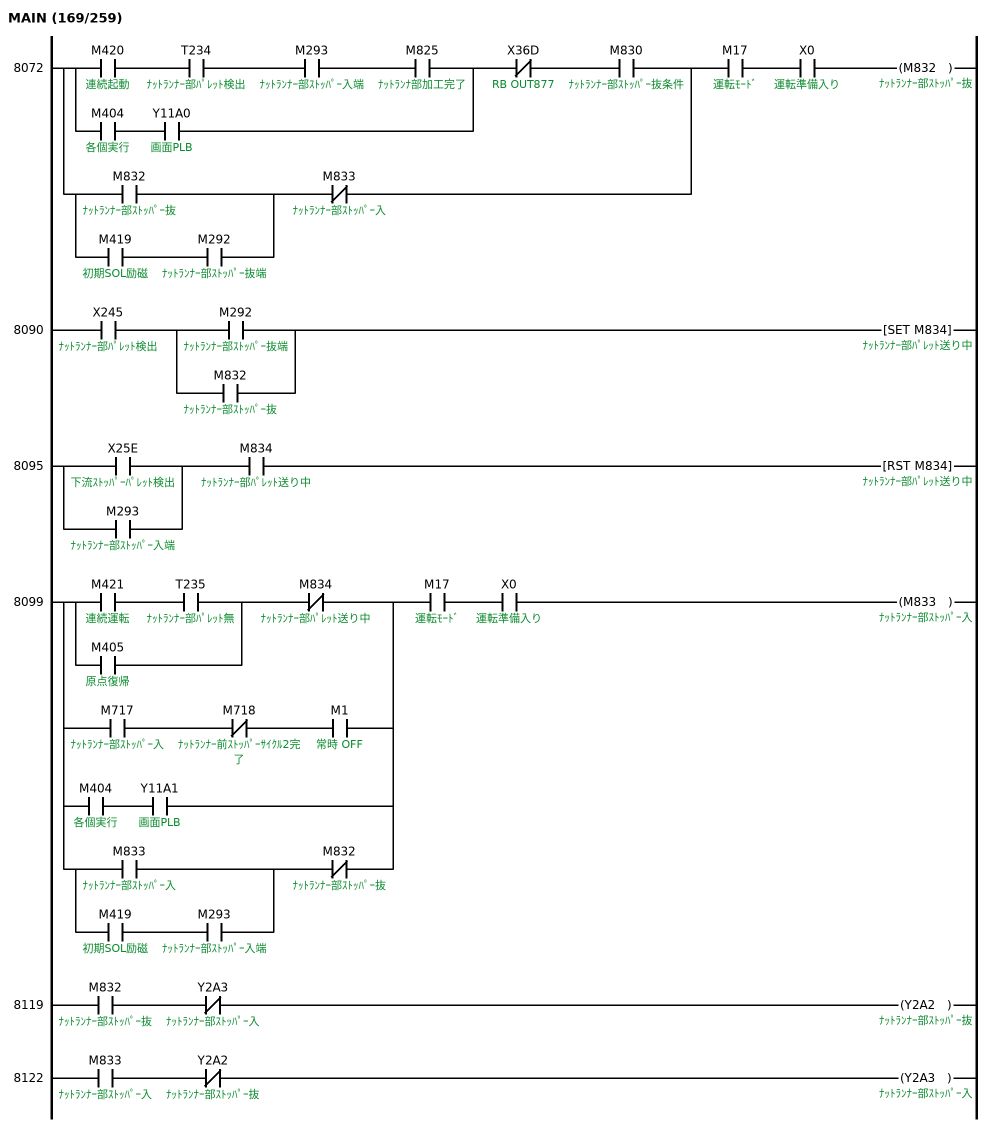
[picture p168: ladder of MAIN, rungs at steps 8072 to 8122]
8072  LD      M420  ; 連続起動
      AND     T234  ; ﾅｯﾄﾗﾝﾅｰ部ﾊﾟﾚｯﾄ検出
      AND     M293  ; ﾅｯﾄﾗﾝﾅｰ部ｽﾄｯﾊﾟｰ入端
      AND     M825  ; ﾅｯﾄﾗﾝﾅ部加工完了
      LD      M404  ; 各個実行
      AND     Y11A0  ; 画面PLB
      ORB
      ANI     X36D  ; RB OUT877
      AND     M830  ; ﾅｯﾄﾗﾝﾅｰ部ｽﾄｯﾊﾟｰ抜条件
      LD      M832  ; ﾅｯﾄﾗﾝﾅｰ部ｽﾄｯﾊﾟｰ抜
      LD      M419  ; 初期SOL励磁
      AND     M292  ; ﾅｯﾄﾗﾝﾅｰ部ｽﾄｯﾊﾟｰ抜端
      ORB
      ANI     M833  ; ﾅｯﾄﾗﾝﾅｰ部ｽﾄｯﾊﾟｰ入
      ORB
      AND     M17  ; 運転ﾓｰﾄﾞ
      AND     X0  ; 運転準備入り
      OUT     M832  ; ﾅｯﾄﾗﾝﾅｰ部ｽﾄｯﾊﾟｰ抜
8090  LD      X245  ; ﾅｯﾄﾗﾝﾅｰ部ﾊﾟﾚｯﾄ検出
      LD      M292  ; ﾅｯﾄﾗﾝﾅｰ部ｽﾄｯﾊﾟｰ抜端
      OR      M832  ; ﾅｯﾄﾗﾝﾅｰ部ｽﾄｯﾊﾟｰ抜
      ANB
      SET     M834  ; ﾅｯﾄﾗﾝﾅｰ部ﾊﾟﾚｯﾄ送り中
8095  LD      X25E  ; 下流ｽﾄｯﾊﾟｰﾊﾟﾚｯﾄ検出
      OR      M293  ; ﾅｯﾄﾗﾝﾅｰ部ｽﾄｯﾊﾟｰ入端
      AND     M834  ; ﾅｯﾄﾗﾝﾅｰ部ﾊﾟﾚｯﾄ送り中
      RST     M834  ; ﾅｯﾄﾗﾝﾅｰ部ﾊﾟﾚｯﾄ送り中
8099  LD      M421  ; 連続運転
      AND     T235  ; ﾅｯﾄﾗﾝﾅｰ部ﾊﾟﾚｯﾄ無
      OR      M405  ; 原点復帰
      ANI     M834  ; ﾅｯﾄﾗﾝﾅｰ部ﾊﾟﾚｯﾄ送り中
      LD      M717  ; ﾅｯﾄﾗﾝﾅｰ部ｽﾄｯﾊﾟｰ入
      ANI     M718  ; ﾅｯﾄﾗﾝﾅｰ前ｽﾄｯﾊﾟｰｻｲｸﾙ2完了
      AND     M1  ; 常時 OFF
      ORB
      LD      M404  ; 各個実行
      AND     Y11A1  ; 画面PLB
      ORB
      LD      M833  ; ﾅｯﾄﾗﾝﾅｰ部ｽﾄｯﾊﾟｰ入
      LD      M419  ; 初期SOL励磁
      AND     M293  ; ﾅｯﾄﾗﾝﾅｰ部ｽﾄｯﾊﾟｰ入端
      ORB
      ANI     M832  ; ﾅｯﾄﾗﾝﾅｰ部ｽﾄｯﾊﾟｰ抜
      ORB
      AND     M17  ; 運転ﾓｰﾄﾞ
      AND     X0  ; 運転準備入り
      OUT     M833  ; ﾅｯﾄﾗﾝﾅｰ部ｽﾄｯﾊﾟｰ入
8119  LD      M832  ; ﾅｯﾄﾗﾝﾅｰ部ｽﾄｯﾊﾟｰ抜
      ANI     Y2A3  ; ﾅｯﾄﾗﾝﾅｰ部ｽﾄｯﾊﾟｰ入
      OUT     Y2A2  ; ﾅｯﾄﾗﾝﾅｰ部ｽﾄｯﾊﾟｰ抜
8122  LD      M833  ; ﾅｯﾄﾗﾝﾅｰ部ｽﾄｯﾊﾟｰ入
      ANI     Y2A2  ; ﾅｯﾄﾗﾝﾅｰ部ｽﾄｯﾊﾟｰ抜
      OUT     Y2A3  ; ﾅｯﾄﾗﾝﾅｰ部ｽﾄｯﾊﾟｰ入
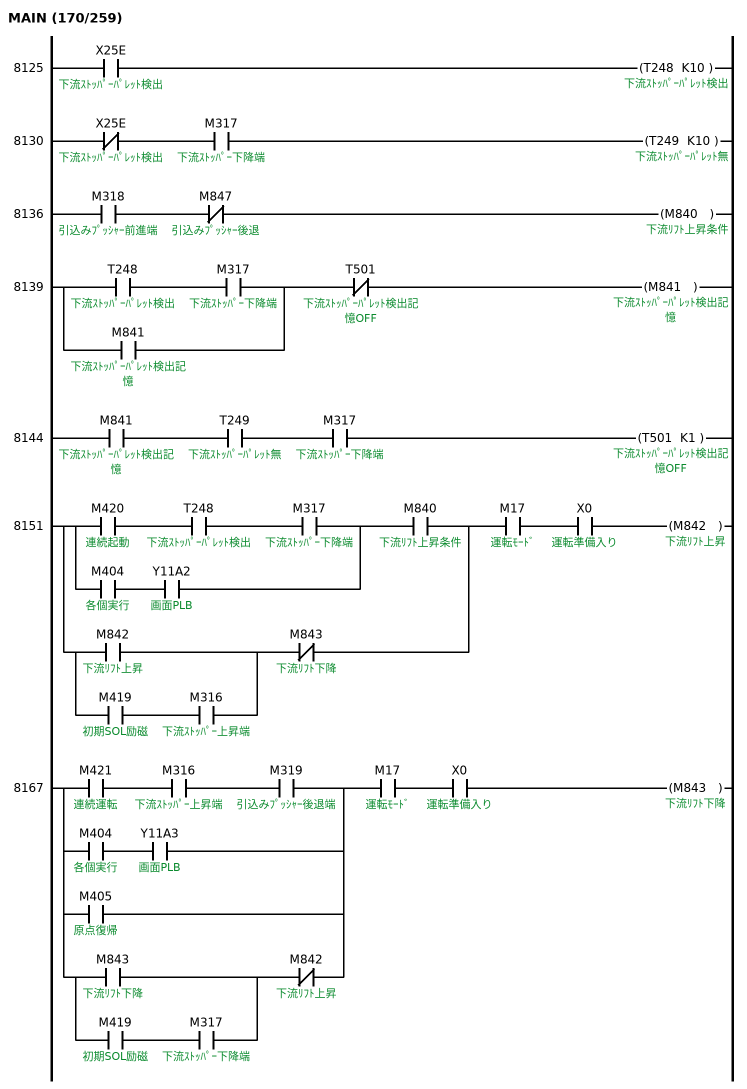
8125  LD      X25E  ; 下流ｽﾄｯﾊﾟｰﾊﾟﾚｯﾄ検出
      OUT     T248 K10  ; 下流ｽﾄｯﾊﾟｰﾊﾟﾚｯﾄ検出
8130  LDI     X25E  ; 下流ｽﾄｯﾊﾟｰﾊﾟﾚｯﾄ検出
      AND     M317  ; 下流ｽﾄｯﾊﾟｰ下降端
      OUT     T249 K10  ; 下流ｽﾄｯﾊﾟｰﾊﾟﾚｯﾄ無
8136  LD      M318  ; 引込みﾌﾟｯｼｬｰ前進端
      ANI     M847  ; 引込みﾌﾟｯｼｬｰ後退
      OUT     M840  ; 下流ﾘﾌﾄ上昇条件
8139  LD      T248  ; 下流ｽﾄｯﾊﾟｰﾊﾟﾚｯﾄ検出
      AND     M317  ; 下流ｽﾄｯﾊﾟｰ下降端
      OR      M841  ; 下流ｽﾄｯﾊﾟｰﾊﾟﾚｯﾄ検出記憶
      ANI     T501  ; 下流ｽﾄｯﾊﾟｰﾊﾟﾚｯﾄ検出記憶OFF
      OUT     M841  ; 下流ｽﾄｯﾊﾟｰﾊﾟﾚｯﾄ検出記憶
8144  LD      M841  ; 下流ｽﾄｯﾊﾟｰﾊﾟﾚｯﾄ検出記憶
      AND     T249  ; 下流ｽﾄｯﾊﾟｰﾊﾟﾚｯﾄ無
      AND     M317  ; 下流ｽﾄｯﾊﾟｰ下降端
      OUT     T501 K1  ; 下流ｽﾄｯﾊﾟｰﾊﾟﾚｯﾄ検出記憶OFF
8151  LD      M420  ; 連続起動
      AND     T248  ; 下流ｽﾄｯﾊﾟｰﾊﾟﾚｯﾄ検出
      AND     M317  ; 下流ｽﾄｯﾊﾟｰ下降端
      LD      M404  ; 各個実行
      AND     Y11A2  ; 画面PLB
      ORB
      AND     M840  ; 下流ﾘﾌﾄ上昇条件
      LD      M842  ; 下流ﾘﾌﾄ上昇
      LD      M419  ; 初期SOL励磁
      AND     M316  ; 下流ｽﾄｯﾊﾟｰ上昇端
      ORB
      ANI     M843  ; 下流ﾘﾌﾄ下降
      ORB
      AND     M17  ; 運転ﾓｰﾄﾞ
      AND     X0  ; 運転準備入り
      OUT     M842  ; 下流ﾘﾌﾄ上昇
8167  LD      M421  ; 連続運転
      AND     M316  ; 下流ｽﾄｯﾊﾟｰ上昇端
      AND     M319  ; 引込みﾌﾟｯｼｬｰ後退端
      LD      M404  ; 各個実行
      AND     Y11A3  ; 画面PLB
      ORB
      OR      M405  ; 原点復帰
      LD      M843  ; 下流ﾘﾌﾄ下降
      LD      M419  ; 初期SOL励磁
      AND     M317  ; 下流ｽﾄｯﾊﾟｰ下降端
      ORB
      ANI     M842  ; 下流ﾘﾌﾄ上昇
      ORB
      AND     M17  ; 運転ﾓｰﾄﾞ
      AND     X0  ; 運転準備入り
      OUT     M843  ; 下流ﾘﾌﾄ下降
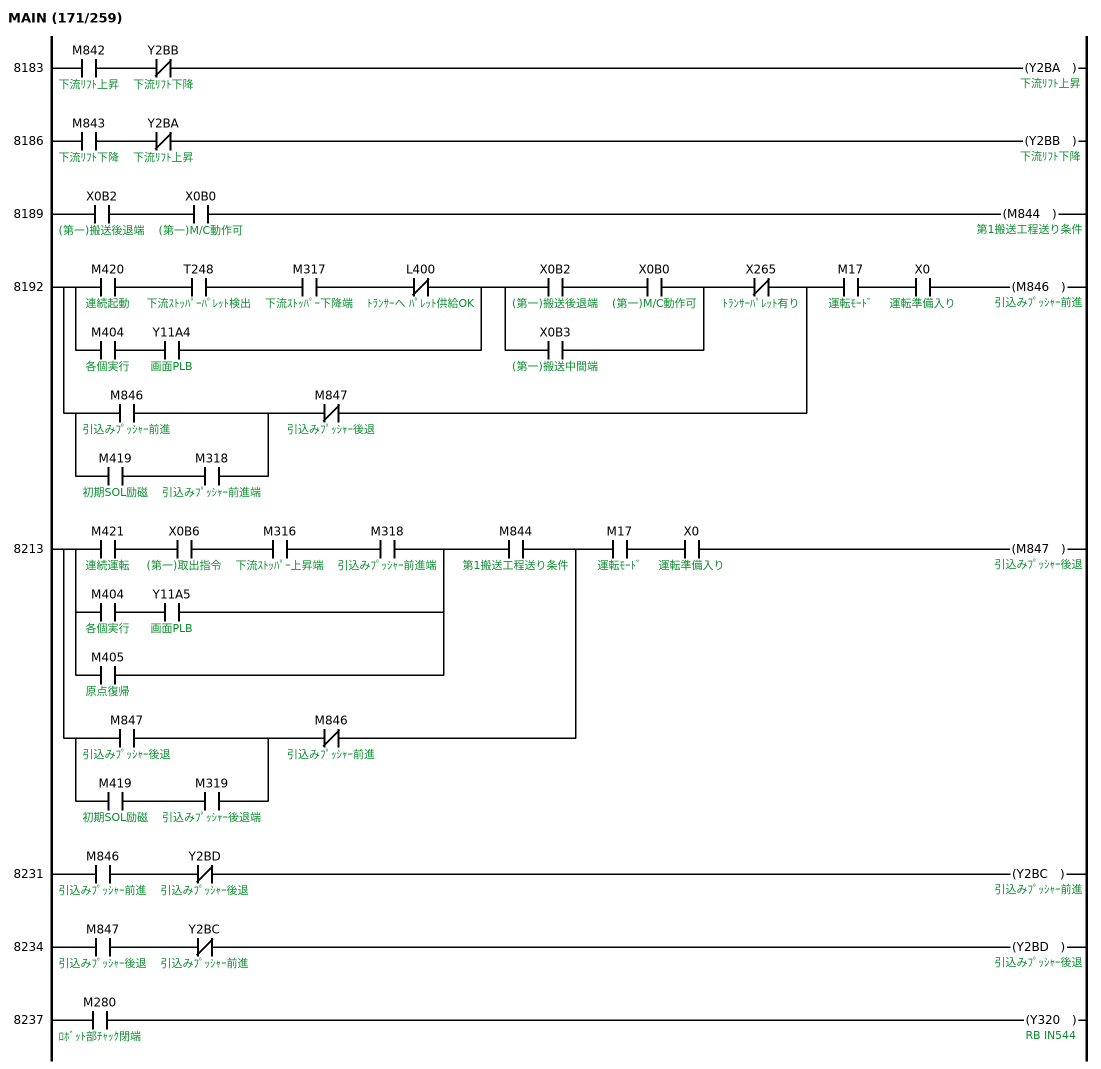
8183  LD      M842  ; 下流ﾘﾌﾄ上昇
      ANI     Y2BB  ; 下流ﾘﾌﾄ下降
      OUT     Y2BA  ; 下流ﾘﾌﾄ上昇
8186  LD      M843  ; 下流ﾘﾌﾄ下降
      ANI     Y2BA  ; 下流ﾘﾌﾄ上昇
      OUT     Y2BB  ; 下流ﾘﾌﾄ下降
8189  LD      X0B2  ; (第一)搬送後退端
      AND     X0B0  ; (第一)M/C動作可
      OUT     M844  ; 第1搬送工程送り条件
8192  LD      M420  ; 連続起動
      AND     T248  ; 下流ｽﾄｯﾊﾟｰﾊﾟﾚｯﾄ検出
      AND     M317  ; 下流ｽﾄｯﾊﾟｰ下降端
      ANI     L400  ; ﾄﾗﾝｻｰへ ﾊﾟﾚｯﾄ供給OK
      LD      M404  ; 各個実行
      AND     Y11A4  ; 画面PLB
      ORB
      LD      X0B2  ; (第一)搬送後退端
      AND     X0B0  ; (第一)M/C動作可
      OR      X0B3  ; (第一)搬送中間端
      ANB
      ANI     X265  ; ﾄﾗﾝｻｰﾊﾟﾚｯﾄ有り
      LD      M846  ; 引込みﾌﾟｯｼｬｰ前進
      LD      M419  ; 初期SOL励磁
      AND     M318  ; 引込みﾌﾟｯｼｬｰ前進端
      ORB
      ANI     M847  ; 引込みﾌﾟｯｼｬｰ後退
      ORB
      AND     M17  ; 運転ﾓｰﾄﾞ
      AND     X0  ; 運転準備入り
      OUT     M846  ; 引込みﾌﾟｯｼｬｰ前進
8213  LD      M421  ; 連続運転
      AND     X0B6  ; (第一)取出指令
      AND     M316  ; 下流ｽﾄｯﾊﾟｰ上昇端
      AND     M318  ; 引込みﾌﾟｯｼｬｰ前進端
      LD      M404  ; 各個実行
      AND     Y11A5  ; 画面PLB
      ORB
      OR      M405  ; 原点復帰
      AND     M844  ; 第1搬送工程送り条件
      LD      M847  ; 引込みﾌﾟｯｼｬｰ後退
      LD      M419  ; 初期SOL励磁
      AND     M319  ; 引込みﾌﾟｯｼｬｰ後退端
      ORB
      ANI     M846  ; 引込みﾌﾟｯｼｬｰ前進
      ORB
      AND     M17  ; 運転ﾓｰﾄﾞ
      AND     X0  ; 運転準備入り
      OUT     M847  ; 引込みﾌﾟｯｼｬｰ後退
8231  LD      M846  ; 引込みﾌﾟｯｼｬｰ前進
      ANI     Y2BD  ; 引込みﾌﾟｯｼｬｰ後退
      OUT     Y2BC  ; 引込みﾌﾟｯｼｬｰ前進
8234  LD      M847  ; 引込みﾌﾟｯｼｬｰ後退
      ANI     Y2BC  ; 引込みﾌﾟｯｼｬｰ前進
      OUT     Y2BD  ; 引込みﾌﾟｯｼｬｰ後退
8237  LD      M280  ; ﾛﾎﾞｯﾄ部ﾁｬｯｸ閉端
      OUT     Y320  ; RB IN544
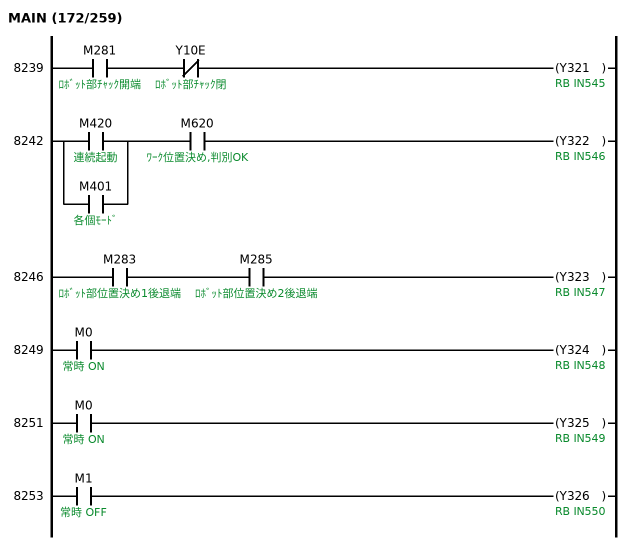
8239  LD      M281  ; ﾛﾎﾞｯﾄ部ﾁｬｯｸ開端
      ANI     Y10E  ; ﾛﾎﾞｯﾄ部ﾁｬｯｸ閉
      OUT     Y321  ; RB IN545
8242  LD      M420  ; 連続起動
      OR      M401  ; 各個ﾓｰﾄﾞ
      AND     M620  ; ﾜｰｸ位置決め,判別OK
      OUT     Y322  ; RB IN546
8246  LD      M283  ; ﾛﾎﾞｯﾄ部位置決め1後退端
      AND     M285  ; ﾛﾎﾞｯﾄ部位置決め2後退端
      OUT     Y323  ; RB IN547
8249  LD      M0  ; 常時 ON
      OUT     Y324  ; RB IN548
8251  LD      M0  ; 常時 ON
      OUT     Y325  ; RB IN549
8253  LD      M1  ; 常時 OFF
      OUT     Y326  ; RB IN550
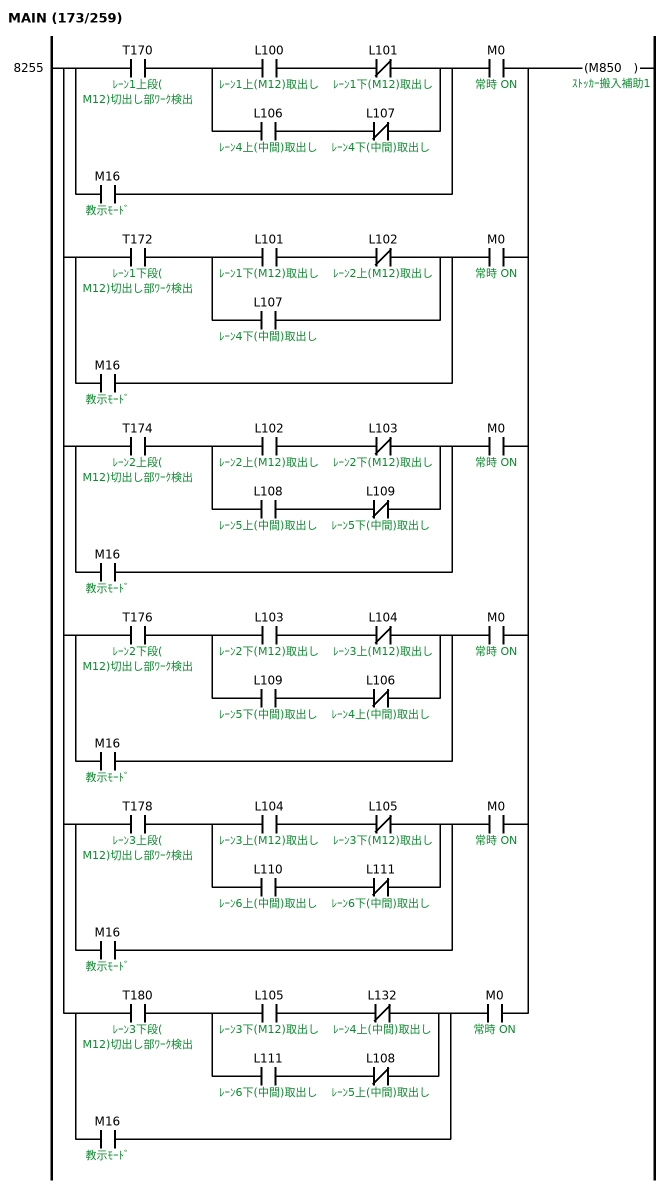
8255  LD      T170  ; ﾚｰﾝ1上段(M12)切出し部ﾜｰｸ検出
      LD      L100  ; ﾚｰﾝ1上(M12)取出し
      ANI     L101  ; ﾚｰﾝ1下(M12)取出し
      LD      L106  ; ﾚｰﾝ4上(中間)取出し
      ANI     L107  ; ﾚｰﾝ4下(中間)取出し
      ORB
      ANB
      OR      M16  ; 教示ﾓｰﾄﾞ
      AND     M0  ; 常時 ON
      LD      T172  ; ﾚｰﾝ1下段(M12)切出し部ﾜｰｸ検出
      LD      L101  ; ﾚｰﾝ1下(M12)取出し
      ANI     L102  ; ﾚｰﾝ2上(M12)取出し
      OR      L107  ; ﾚｰﾝ4下(中間)取出し
      ANB
      OR      M16  ; 教示ﾓｰﾄﾞ
      AND     M0  ; 常時 ON
      ORB
      LD      T174  ; ﾚｰﾝ2上段(M12)切出し部ﾜｰｸ検出
      LD      L102  ; ﾚｰﾝ2上(M12)取出し
      ANI     L103  ; ﾚｰﾝ2下(M12)取出し
      LD      L108  ; ﾚｰﾝ5上(中間)取出し
      ANI     L109  ; ﾚｰﾝ5下(中間)取出し
      ORB
      ANB
      OR      M16  ; 教示ﾓｰﾄﾞ
      AND     M0  ; 常時 ON
      ORB
      LD      T176  ; ﾚｰﾝ2下段(M12)切出し部ﾜｰｸ検出
      LD      L103  ; ﾚｰﾝ2下(M12)取出し
      ANI     L104  ; ﾚｰﾝ3上(M12)取出し
      LD      L109  ; ﾚｰﾝ5下(中間)取出し
      ANI     L106  ; ﾚｰﾝ4上(中間)取出し
      ORB
      ANB
      OR      M16  ; 教示ﾓｰﾄﾞ
      AND     M0  ; 常時 ON
      ORB
      LD      T178  ; ﾚｰﾝ3上段(M12)切出し部ﾜｰｸ検出
      LD      L104  ; ﾚｰﾝ3上(M12)取出し
      ANI     L105  ; ﾚｰﾝ3下(M12)取出し
      LD      L110  ; ﾚｰﾝ6上(中間)取出し
      ANI     L111  ; ﾚｰﾝ6下(中間)取出し
      ORB
      ANB
      OR      M16  ; 教示ﾓｰﾄﾞ
      AND     M0  ; 常時 ON
      ORB
      LD      T180  ; ﾚｰﾝ3下段(M12)切出し部ﾜｰｸ検出
      LD      L105  ; ﾚｰﾝ3下(M12)取出し
      ANI     L132  ; ﾚｰﾝ4上(中間)取出し
      LD      L111  ; ﾚｰﾝ6下(中間)取出し
      ANI     L108  ; ﾚｰﾝ5上(中間)取出し
      ORB
      ANB
      OR      M16  ; 教示ﾓｰﾄﾞ
      AND     M0  ; 常時 ON
      ORB
      OUT     M850  ; ｽﾄｯｶｰ搬入補助1
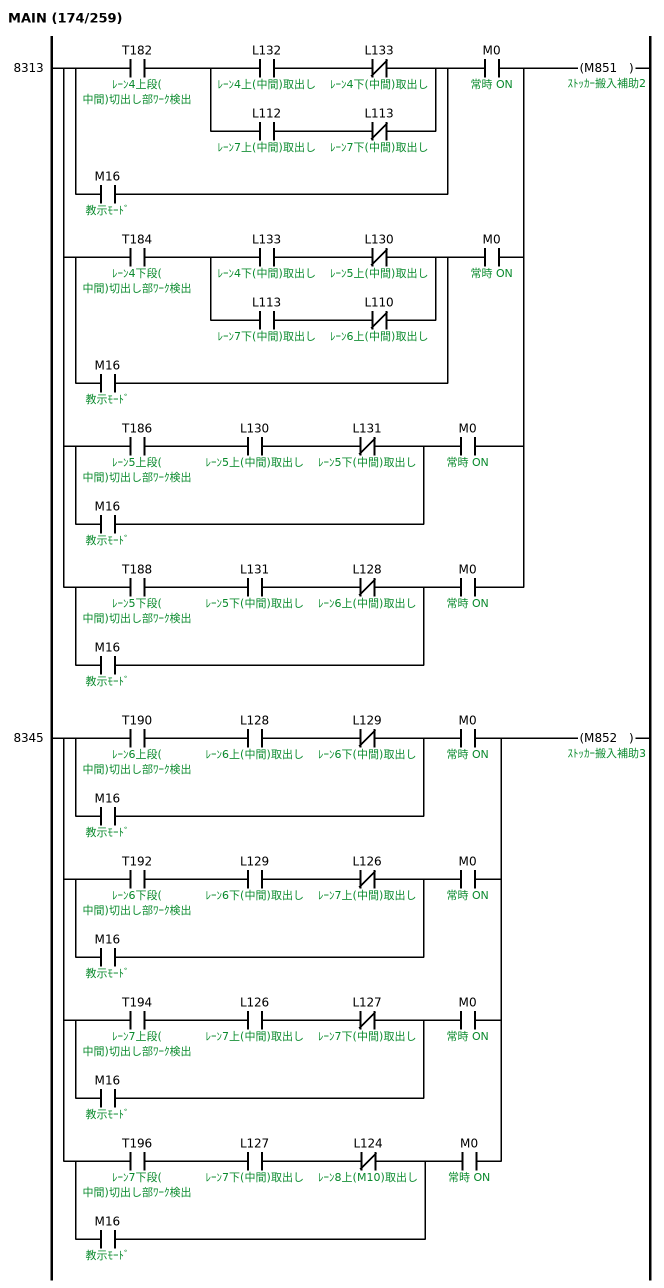
8313  LD      T182  ; ﾚｰﾝ4上段(中間)切出し部ﾜｰｸ検出
      LD      L132  ; ﾚｰﾝ4上(中間)取出し
      ANI     L133  ; ﾚｰﾝ4下(中間)取出し
      LD      L112  ; ﾚｰﾝ7上(中間)取出し
      ANI     L113  ; ﾚｰﾝ7下(中間)取出し
      ORB
      ANB
      OR      M16  ; 教示ﾓｰﾄﾞ
      AND     M0  ; 常時 ON
      LD      T184  ; ﾚｰﾝ4下段(中間)切出し部ﾜｰｸ検出
      LD      L133  ; ﾚｰﾝ4下(中間)取出し
      ANI     L130  ; ﾚｰﾝ5上(中間)取出し
      LD      L113  ; ﾚｰﾝ7下(中間)取出し
      ANI     L110  ; ﾚｰﾝ6上(中間)取出し
      ORB
      ANB
      OR      M16  ; 教示ﾓｰﾄﾞ
      AND     M0  ; 常時 ON
      ORB
      LD      T186  ; ﾚｰﾝ5上段(中間)切出し部ﾜｰｸ検出
      AND     L130  ; ﾚｰﾝ5上(中間)取出し
      ANI     L131  ; ﾚｰﾝ5下(中間)取出し
      OR      M16  ; 教示ﾓｰﾄﾞ
      AND     M0  ; 常時 ON
      ORB
      LD      T188  ; ﾚｰﾝ5下段(中間)切出し部ﾜｰｸ検出
      AND     L131  ; ﾚｰﾝ5下(中間)取出し
      ANI     L128  ; ﾚｰﾝ6上(中間)取出し
      OR      M16  ; 教示ﾓｰﾄﾞ
      AND     M0  ; 常時 ON
      ORB
      OUT     M851  ; ｽﾄｯｶｰ搬入補助2
8345  LD      T190  ; ﾚｰﾝ6上段(中間)切出し部ﾜｰｸ検出
      AND     L128  ; ﾚｰﾝ6上(中間)取出し
      ANI     L129  ; ﾚｰﾝ6下(中間)取出し
      OR      M16  ; 教示ﾓｰﾄﾞ
      AND     M0  ; 常時 ON
      LD      T192  ; ﾚｰﾝ6下段(中間)切出し部ﾜｰｸ検出
      AND     L129  ; ﾚｰﾝ6下(中間)取出し
      ANI     L126  ; ﾚｰﾝ7上(中間)取出し
      OR      M16  ; 教示ﾓｰﾄﾞ
      AND     M0  ; 常時 ON
      ORB
      LD      T194  ; ﾚｰﾝ7上段(中間)切出し部ﾜｰｸ検出
      AND     L126  ; ﾚｰﾝ7上(中間)取出し
      ANI     L127  ; ﾚｰﾝ7下(中間)取出し
      OR      M16  ; 教示ﾓｰﾄﾞ
      AND     M0  ; 常時 ON
      ORB
      LD      T196  ; ﾚｰﾝ7下段(中間)切出し部ﾜｰｸ検出
      AND     L127  ; ﾚｰﾝ7下(中間)取出し
      ANI     L124  ; ﾚｰﾝ8上(M10)取出し
      OR      M16  ; 教示ﾓｰﾄﾞ
      AND     M0  ; 常時 ON
      ORB
      OUT     M852  ; ｽﾄｯｶｰ搬入補助3
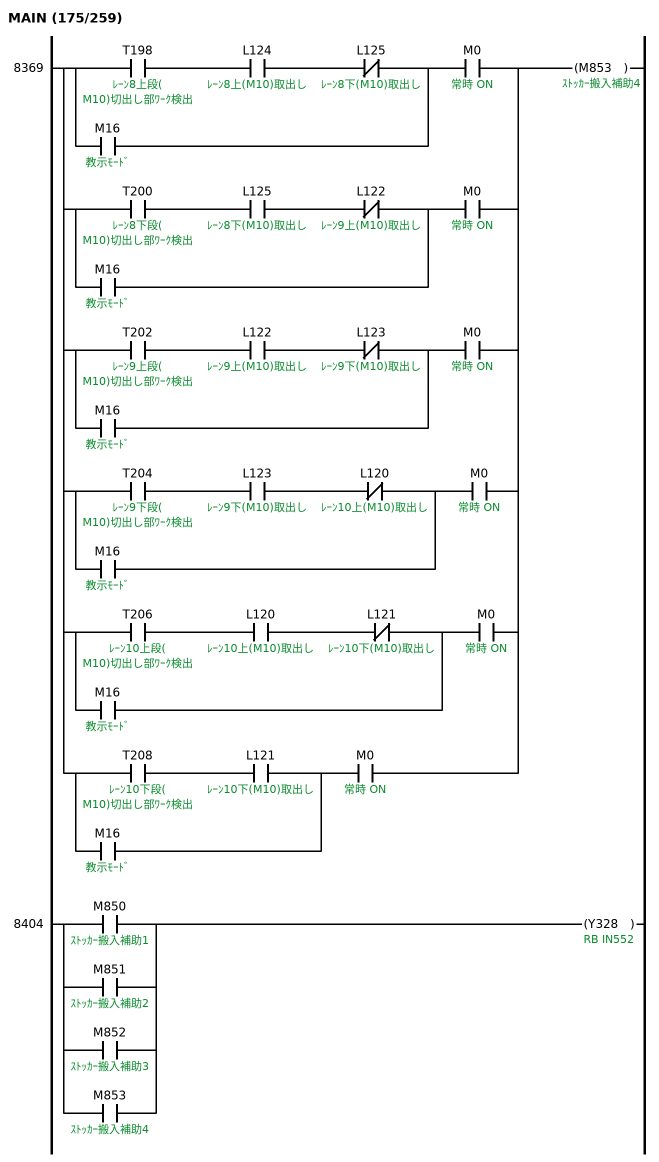
8369  LD      T198  ; ﾚｰﾝ8上段(M10)切出し部ﾜｰｸ検出
      AND     L124  ; ﾚｰﾝ8上(M10)取出し
      ANI     L125  ; ﾚｰﾝ8下(M10)取出し
      OR      M16  ; 教示ﾓｰﾄﾞ
      AND     M0  ; 常時 ON
      LD      T200  ; ﾚｰﾝ8下段(M10)切出し部ﾜｰｸ検出
      AND     L125  ; ﾚｰﾝ8下(M10)取出し
      ANI     L122  ; ﾚｰﾝ9上(M10)取出し
      OR      M16  ; 教示ﾓｰﾄﾞ
      AND     M0  ; 常時 ON
      ORB
      LD      T202  ; ﾚｰﾝ9上段(M10)切出し部ﾜｰｸ検出
      AND     L122  ; ﾚｰﾝ9上(M10)取出し
      ANI     L123  ; ﾚｰﾝ9下(M10)取出し
      OR      M16  ; 教示ﾓｰﾄﾞ
      AND     M0  ; 常時 ON
      ORB
      LD      T204  ; ﾚｰﾝ9下段(M10)切出し部ﾜｰｸ検出
      AND     L123  ; ﾚｰﾝ9下(M10)取出し
      ANI     L120  ; ﾚｰﾝ10上(M10)取出し
      OR      M16  ; 教示ﾓｰﾄﾞ
      AND     M0  ; 常時 ON
      ORB
      LD      T206  ; ﾚｰﾝ10上段(M10)切出し部ﾜｰｸ検出
      AND     L120  ; ﾚｰﾝ10上(M10)取出し
      ANI     L121  ; ﾚｰﾝ10下(M10)取出し
      OR      M16  ; 教示ﾓｰﾄﾞ
      AND     M0  ; 常時 ON
      ORB
      LD      T208  ; ﾚｰﾝ10下段(M10)切出し部ﾜｰｸ検出
      AND     L121  ; ﾚｰﾝ10下(M10)取出し
      OR      M16  ; 教示ﾓｰﾄﾞ
      AND     M0  ; 常時 ON
      ORB
      OUT     M853  ; ｽﾄｯｶｰ搬入補助4
8404  LD      M850  ; ｽﾄｯｶｰ搬入補助1
      OR      M851  ; ｽﾄｯｶｰ搬入補助2
      OR      M852  ; ｽﾄｯｶｰ搬入補助3
      OR      M853  ; ｽﾄｯｶｰ搬入補助4
      OUT     Y328  ; RB IN552
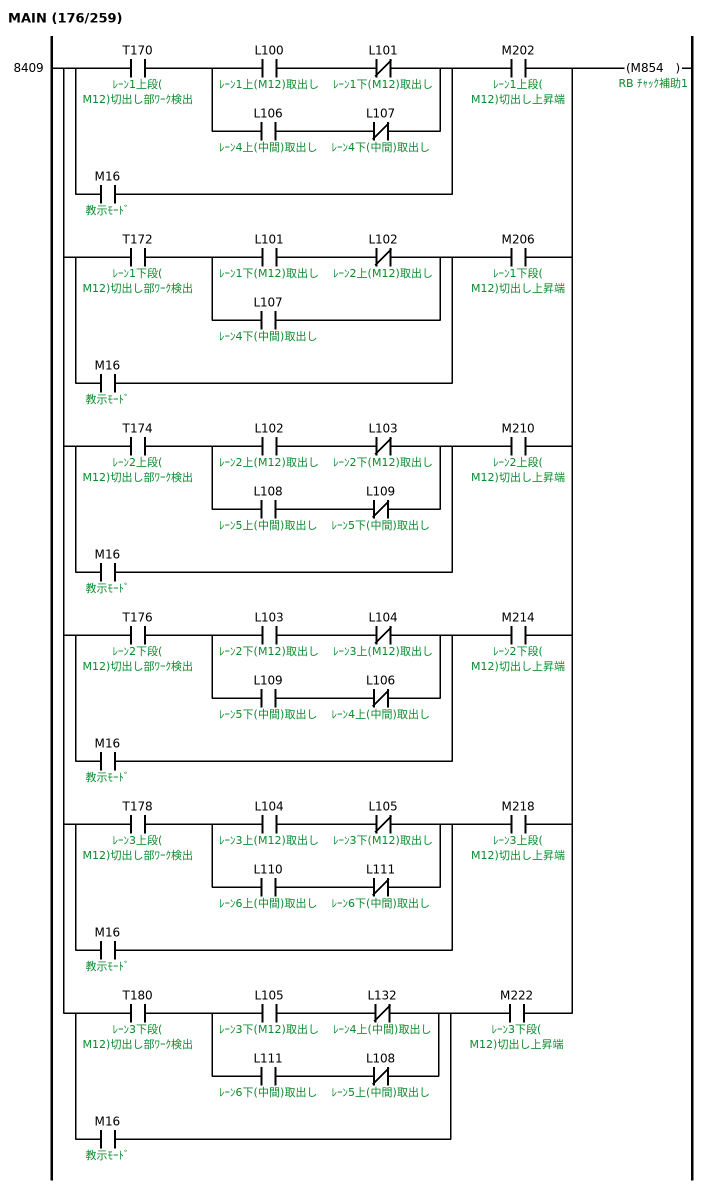
8409  LD      T170  ; ﾚｰﾝ1上段(M12)切出し部ﾜｰｸ検出
      LD      L100  ; ﾚｰﾝ1上(M12)取出し
      ANI     L101  ; ﾚｰﾝ1下(M12)取出し
      LD      L106  ; ﾚｰﾝ4上(中間)取出し
      ANI     L107  ; ﾚｰﾝ4下(中間)取出し
      ORB
      ANB
      OR      M16  ; 教示ﾓｰﾄﾞ
      AND     M202  ; ﾚｰﾝ1上段(M12)切出し上昇端
      LD      T172  ; ﾚｰﾝ1下段(M12)切出し部ﾜｰｸ検出
      LD      L101  ; ﾚｰﾝ1下(M12)取出し
      ANI     L102  ; ﾚｰﾝ2上(M12)取出し
      OR      L107  ; ﾚｰﾝ4下(中間)取出し
      ANB
      OR      M16  ; 教示ﾓｰﾄﾞ
      AND     M206  ; ﾚｰﾝ1下段(M12)切出し上昇端
      ORB
      LD      T174  ; ﾚｰﾝ2上段(M12)切出し部ﾜｰｸ検出
      LD      L102  ; ﾚｰﾝ2上(M12)取出し
      ANI     L103  ; ﾚｰﾝ2下(M12)取出し
      LD      L108  ; ﾚｰﾝ5上(中間)取出し
      ANI     L109  ; ﾚｰﾝ5下(中間)取出し
      ORB
      ANB
      OR      M16  ; 教示ﾓｰﾄﾞ
      AND     M210  ; ﾚｰﾝ2上段(M12)切出し上昇端
      ORB
      LD      T176  ; ﾚｰﾝ2下段(M12)切出し部ﾜｰｸ検出
      LD      L103  ; ﾚｰﾝ2下(M12)取出し
      ANI     L104  ; ﾚｰﾝ3上(M12)取出し
      LD      L109  ; ﾚｰﾝ5下(中間)取出し
      ANI     L106  ; ﾚｰﾝ4上(中間)取出し
      ORB
      ANB
      OR      M16  ; 教示ﾓｰﾄﾞ
      AND     M214  ; ﾚｰﾝ2下段(M12)切出し上昇端
      ORB
      LD      T178  ; ﾚｰﾝ3上段(M12)切出し部ﾜｰｸ検出
      LD      L104  ; ﾚｰﾝ3上(M12)取出し
      ANI     L105  ; ﾚｰﾝ3下(M12)取出し
      LD      L110  ; ﾚｰﾝ6上(中間)取出し
      ANI     L111  ; ﾚｰﾝ6下(中間)取出し
      ORB
      ANB
      OR      M16  ; 教示ﾓｰﾄﾞ
      AND     M218  ; ﾚｰﾝ3上段(M12)切出し上昇端
      ORB
      LD      T180  ; ﾚｰﾝ3下段(M12)切出し部ﾜｰｸ検出
      LD      L105  ; ﾚｰﾝ3下(M12)取出し
      ANI     L132  ; ﾚｰﾝ4上(中間)取出し
      LD      L111  ; ﾚｰﾝ6下(中間)取出し
      ANI     L108  ; ﾚｰﾝ5上(中間)取出し
      ORB
      ANB
      OR      M16  ; 教示ﾓｰﾄﾞ
      AND     M222  ; ﾚｰﾝ3下段(M12)切出し上昇端
      ORB
      OUT     M854  ; RB ﾁｬｯｸ補助1
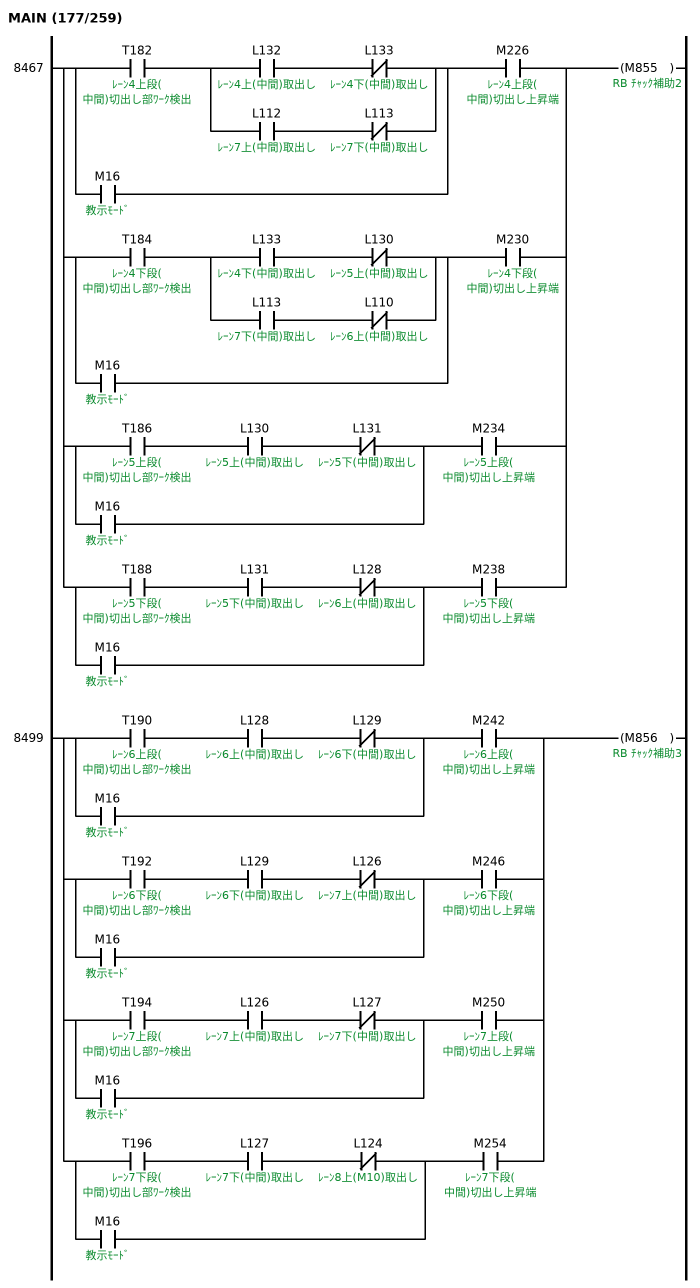
8467  LD      T182  ; ﾚｰﾝ4上段(中間)切出し部ﾜｰｸ検出
      LD      L132  ; ﾚｰﾝ4上(中間)取出し
      ANI     L133  ; ﾚｰﾝ4下(中間)取出し
      LD      L112  ; ﾚｰﾝ7上(中間)取出し
      ANI     L113  ; ﾚｰﾝ7下(中間)取出し
      ORB
      ANB
      OR      M16  ; 教示ﾓｰﾄﾞ
      AND     M226  ; ﾚｰﾝ4上段(中間)切出し上昇端
      LD      T184  ; ﾚｰﾝ4下段(中間)切出し部ﾜｰｸ検出
      LD      L133  ; ﾚｰﾝ4下(中間)取出し
      ANI     L130  ; ﾚｰﾝ5上(中間)取出し
      LD      L113  ; ﾚｰﾝ7下(中間)取出し
      ANI     L110  ; ﾚｰﾝ6上(中間)取出し
      ORB
      ANB
      OR      M16  ; 教示ﾓｰﾄﾞ
      AND     M230  ; ﾚｰﾝ4下段(中間)切出し上昇端
      ORB
      LD      T186  ; ﾚｰﾝ5上段(中間)切出し部ﾜｰｸ検出
      AND     L130  ; ﾚｰﾝ5上(中間)取出し
      ANI     L131  ; ﾚｰﾝ5下(中間)取出し
      OR      M16  ; 教示ﾓｰﾄﾞ
      AND     M234  ; ﾚｰﾝ5上段(中間)切出し上昇端
      ORB
      LD      T188  ; ﾚｰﾝ5下段(中間)切出し部ﾜｰｸ検出
      AND     L131  ; ﾚｰﾝ5下(中間)取出し
      ANI     L128  ; ﾚｰﾝ6上(中間)取出し
      OR      M16  ; 教示ﾓｰﾄﾞ
      AND     M238  ; ﾚｰﾝ5下段(中間)切出し上昇端
      ORB
      OUT     M855  ; RB ﾁｬｯｸ補助2
8499  LD      T190  ; ﾚｰﾝ6上段(中間)切出し部ﾜｰｸ検出
      AND     L128  ; ﾚｰﾝ6上(中間)取出し
      ANI     L129  ; ﾚｰﾝ6下(中間)取出し
      OR      M16  ; 教示ﾓｰﾄﾞ
      AND     M242  ; ﾚｰﾝ6上段(中間)切出し上昇端
      LD      T192  ; ﾚｰﾝ6下段(中間)切出し部ﾜｰｸ検出
      AND     L129  ; ﾚｰﾝ6下(中間)取出し
      ANI     L126  ; ﾚｰﾝ7上(中間)取出し
      OR      M16  ; 教示ﾓｰﾄﾞ
      AND     M246  ; ﾚｰﾝ6下段(中間)切出し上昇端
      ORB
      LD      T194  ; ﾚｰﾝ7上段(中間)切出し部ﾜｰｸ検出
      AND     L126  ; ﾚｰﾝ7上(中間)取出し
      ANI     L127  ; ﾚｰﾝ7下(中間)取出し
      OR      M16  ; 教示ﾓｰﾄﾞ
      AND     M250  ; ﾚｰﾝ7上段(中間)切出し上昇端
      ORB
      LD      T196  ; ﾚｰﾝ7下段(中間)切出し部ﾜｰｸ検出
      AND     L127  ; ﾚｰﾝ7下(中間)取出し
      ANI     L124  ; ﾚｰﾝ8上(M10)取出し
      OR      M16  ; 教示ﾓｰﾄﾞ
      AND     M254  ; ﾚｰﾝ7下段(中間)切出し上昇端
      ORB
      OUT     M856  ; RB ﾁｬｯｸ補助3
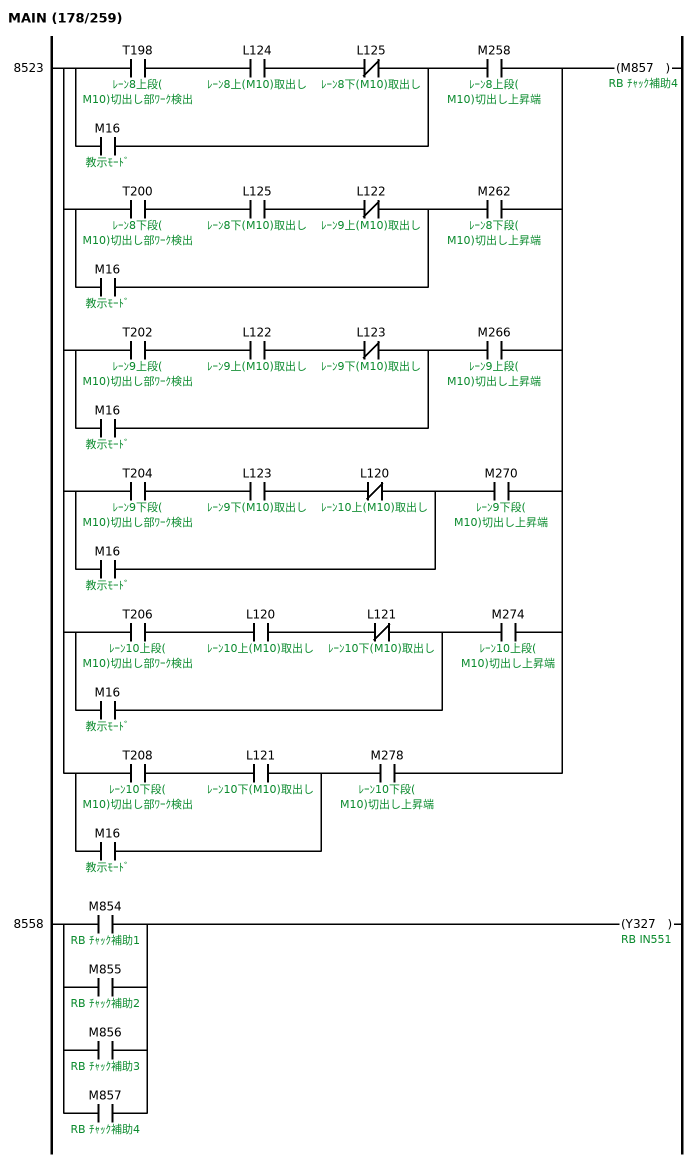
8523  LD      T198  ; ﾚｰﾝ8上段(M10)切出し部ﾜｰｸ検出
      AND     L124  ; ﾚｰﾝ8上(M10)取出し
      ANI     L125  ; ﾚｰﾝ8下(M10)取出し
      OR      M16  ; 教示ﾓｰﾄﾞ
      AND     M258  ; ﾚｰﾝ8上段(M10)切出し上昇端
      LD      T200  ; ﾚｰﾝ8下段(M10)切出し部ﾜｰｸ検出
      AND     L125  ; ﾚｰﾝ8下(M10)取出し
      ANI     L122  ; ﾚｰﾝ9上(M10)取出し
      OR      M16  ; 教示ﾓｰﾄﾞ
      AND     M262  ; ﾚｰﾝ8下段(M10)切出し上昇端
      ORB
      LD      T202  ; ﾚｰﾝ9上段(M10)切出し部ﾜｰｸ検出
      AND     L122  ; ﾚｰﾝ9上(M10)取出し
      ANI     L123  ; ﾚｰﾝ9下(M10)取出し
      OR      M16  ; 教示ﾓｰﾄﾞ
      AND     M266  ; ﾚｰﾝ9上段(M10)切出し上昇端
      ORB
      LD      T204  ; ﾚｰﾝ9下段(M10)切出し部ﾜｰｸ検出
      AND     L123  ; ﾚｰﾝ9下(M10)取出し
      ANI     L120  ; ﾚｰﾝ10上(M10)取出し
      OR      M16  ; 教示ﾓｰﾄﾞ
      AND     M270  ; ﾚｰﾝ9下段(M10)切出し上昇端
      ORB
      LD      T206  ; ﾚｰﾝ10上段(M10)切出し部ﾜｰｸ検出
      AND     L120  ; ﾚｰﾝ10上(M10)取出し
      ANI     L121  ; ﾚｰﾝ10下(M10)取出し
      OR      M16  ; 教示ﾓｰﾄﾞ
      AND     M274  ; ﾚｰﾝ10上段(M10)切出し上昇端
      ORB
      LD      T208  ; ﾚｰﾝ10下段(M10)切出し部ﾜｰｸ検出
      AND     L121  ; ﾚｰﾝ10下(M10)取出し
      OR      M16  ; 教示ﾓｰﾄﾞ
      AND     M278  ; ﾚｰﾝ10下段(M10)切出し上昇端
      ORB
      OUT     M857  ; RB ﾁｬｯｸ補助4
8558  LD      M854  ; RB ﾁｬｯｸ補助1
      OR      M855  ; RB ﾁｬｯｸ補助2
      OR      M856  ; RB ﾁｬｯｸ補助3
      OR      M857  ; RB ﾁｬｯｸ補助4
      OUT     Y327  ; RB IN551
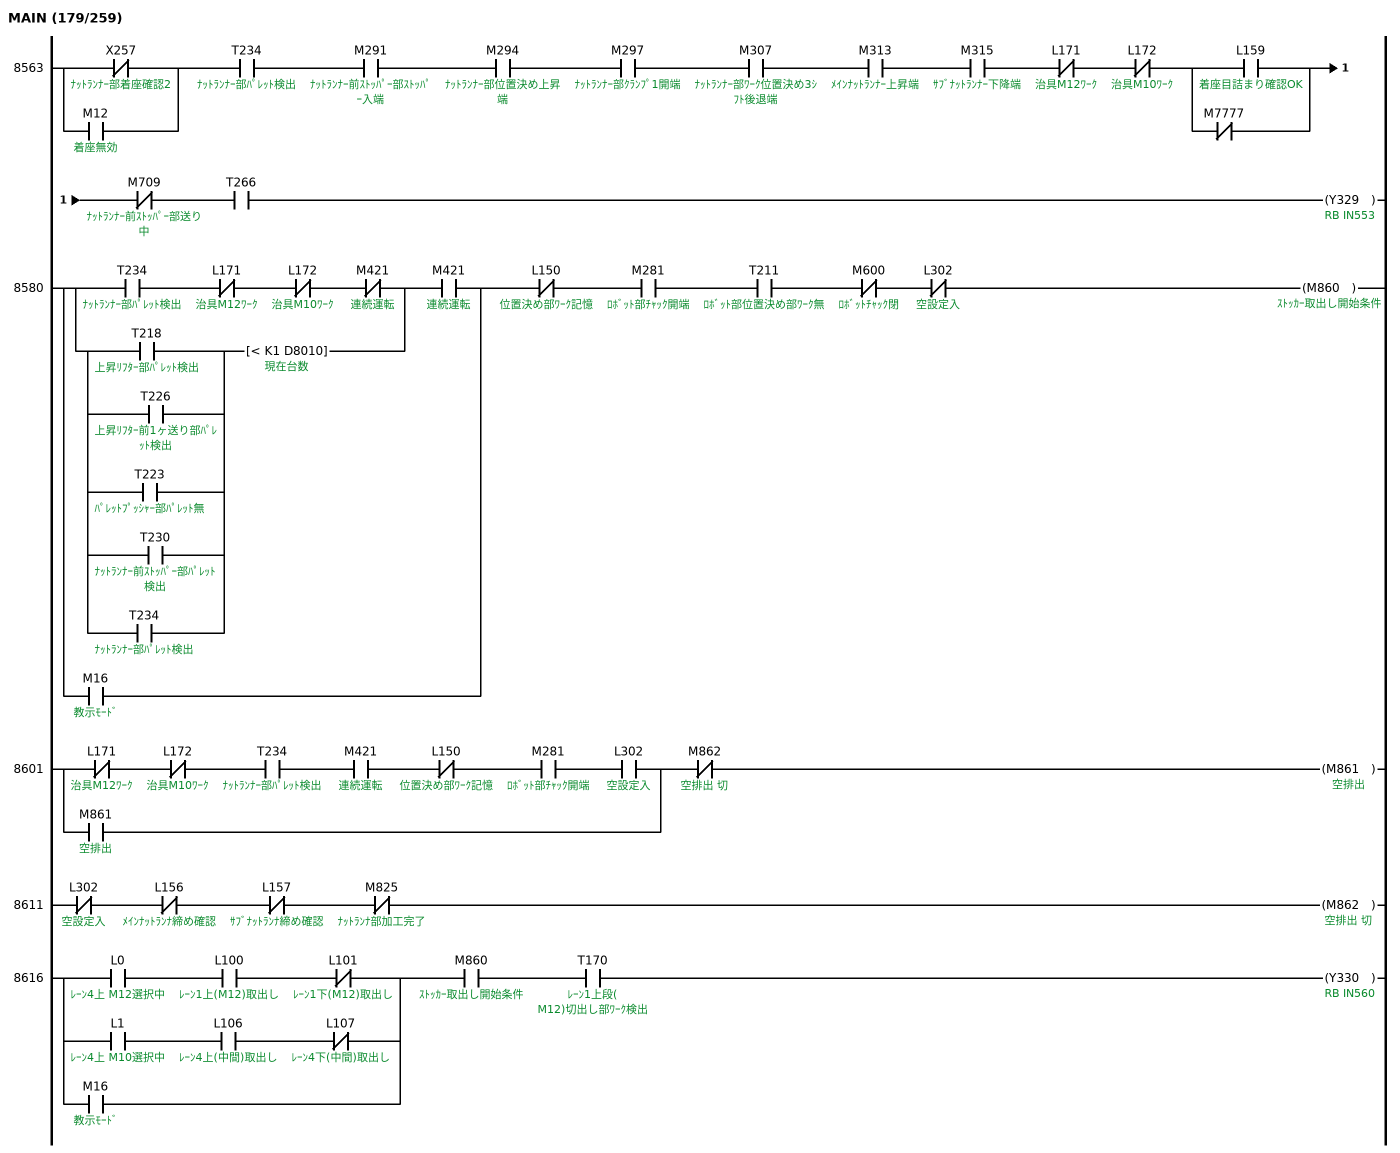
8563  LDI     X257  ; ﾅｯﾄﾗﾝﾅｰ部着座確認2
      OR      M12  ; 着座無効
      AND     T234  ; ﾅｯﾄﾗﾝﾅｰ部ﾊﾟﾚｯﾄ検出
      AND     M291  ; ﾅｯﾄﾗﾝﾅｰ前ｽﾄｯﾊﾟｰ部ｽﾄｯﾊﾟｰ入端
      AND     M294  ; ﾅｯﾄﾗﾝﾅｰ部位置決め上昇端
      AND     M297  ; ﾅｯﾄﾗﾝﾅｰ部ｸﾗﾝﾌﾟ1開端
      AND     M307  ; ﾅｯﾄﾗﾝﾅｰ部ﾜｰｸ位置決め3ｼﾌﾄ後退端
      AND     M313  ; ﾒｲﾝﾅｯﾄﾗﾝﾅｰ上昇端
      AND     M315  ; ｻﾌﾞﾅｯﾄﾗﾝﾅｰ下降端
      ANI     L171  ; 治具M12ﾜｰｸ
      ANI     L172  ; 治具M10ﾜｰｸ
      LD      L159  ; 着座目詰まり確認OK
      ORI     M7777
      ANB
      ANI     M709  ; ﾅｯﾄﾗﾝﾅｰ前ｽﾄｯﾊﾟｰ部送り中
      AND     T266
      OUT     Y329  ; RB IN553
8580  LD      T234  ; ﾅｯﾄﾗﾝﾅｰ部ﾊﾟﾚｯﾄ検出
      ANI     L171  ; 治具M12ﾜｰｸ
      ANI     L172  ; 治具M10ﾜｰｸ
      ANI     M421  ; 連続運転
      LD      T218  ; 上昇ﾘﾌﾀｰ部ﾊﾟﾚｯﾄ検出
      OR      T226  ; 上昇ﾘﾌﾀｰ前1ヶ送り部ﾊﾟﾚｯﾄ検出
      OR      T223  ; ﾊﾟﾚｯﾄﾌﾟｯｼｬｰ部ﾊﾟﾚｯﾄ無
      OR      T230  ; ﾅｯﾄﾗﾝﾅｰ前ｽﾄｯﾊﾟｰ部ﾊﾟﾚｯﾄ検出
      OR      T234  ; ﾅｯﾄﾗﾝﾅｰ部ﾊﾟﾚｯﾄ検出
      AND<    K1 D8010  ; 現在台数
      ORB
      AND     M421  ; 連続運転
      OR      M16  ; 教示ﾓｰﾄﾞ
      ANI     L150  ; 位置決め部ﾜｰｸ記憶
      AND     M281  ; ﾛﾎﾞｯﾄ部ﾁｬｯｸ開端
      AND     T211  ; ﾛﾎﾞｯﾄ部位置決め部ﾜｰｸ無
      ANI     M600  ; ﾛﾎﾞｯﾄﾁｬｯｸ閉
      ANI     L302  ; 空設定入
      OUT     M860  ; ｽﾄｯｶｰ取出し開始条件
8601  LDI     L171  ; 治具M12ﾜｰｸ
      ANI     L172  ; 治具M10ﾜｰｸ
      AND     T234  ; ﾅｯﾄﾗﾝﾅｰ部ﾊﾟﾚｯﾄ検出
      AND     M421  ; 連続運転
      ANI     L150  ; 位置決め部ﾜｰｸ記憶
      AND     M281  ; ﾛﾎﾞｯﾄ部ﾁｬｯｸ開端
      AND     L302  ; 空設定入
      OR      M861  ; 空排出
      ANI     M862  ; 空排出 切
      OUT     M861  ; 空排出
8611  LDI     L302  ; 空設定入
      ANI     L156  ; ﾒｲﾝﾅｯﾄﾗﾝﾅ締め確認
      ANI     L157  ; ｻﾌﾞﾅｯﾄﾗﾝﾅ締め確認
      ANI     M825  ; ﾅｯﾄﾗﾝﾅ部加工完了
      OUT     M862  ; 空排出 切
8616  LD      L0  ; ﾚｰﾝ4上 M12選択中
      AND     L100  ; ﾚｰﾝ1上(M12)取出し
      ANI     L101  ; ﾚｰﾝ1下(M12)取出し
      LD      L1  ; ﾚｰﾝ4上 M10選択中
      AND     L106  ; ﾚｰﾝ4上(中間)取出し
      ANI     L107  ; ﾚｰﾝ4下(中間)取出し
      ORB
      OR      M16  ; 教示ﾓｰﾄﾞ
      AND     M860  ; ｽﾄｯｶｰ取出し開始条件
      AND     T170  ; ﾚｰﾝ1上段(M12)切出し部ﾜｰｸ検出
      OUT     Y330  ; RB IN560
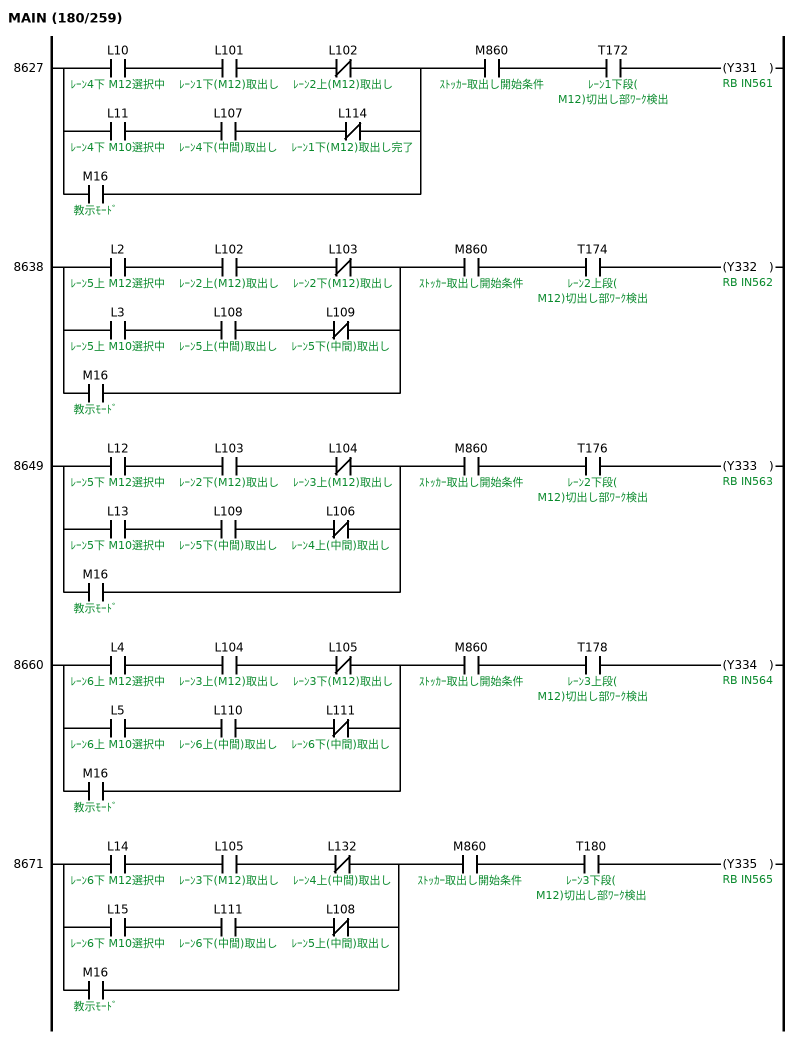
8627  LD      L10  ; ﾚｰﾝ4下 M12選択中
      AND     L101  ; ﾚｰﾝ1下(M12)取出し
      ANI     L102  ; ﾚｰﾝ2上(M12)取出し
      LD      L11  ; ﾚｰﾝ4下 M10選択中
      AND     L107  ; ﾚｰﾝ4下(中間)取出し
      ANI     L114  ; ﾚｰﾝ1下(M12)取出し完了
      ORB
      OR      M16  ; 教示ﾓｰﾄﾞ
      AND     M860  ; ｽﾄｯｶｰ取出し開始条件
      AND     T172  ; ﾚｰﾝ1下段(M12)切出し部ﾜｰｸ検出
      OUT     Y331  ; RB IN561
8638  LD      L2  ; ﾚｰﾝ5上 M12選択中
      AND     L102  ; ﾚｰﾝ2上(M12)取出し
      ANI     L103  ; ﾚｰﾝ2下(M12)取出し
      LD      L3  ; ﾚｰﾝ5上 M10選択中
      AND     L108  ; ﾚｰﾝ5上(中間)取出し
      ANI     L109  ; ﾚｰﾝ5下(中間)取出し
      ORB
      OR      M16  ; 教示ﾓｰﾄﾞ
      AND     M860  ; ｽﾄｯｶｰ取出し開始条件
      AND     T174  ; ﾚｰﾝ2上段(M12)切出し部ﾜｰｸ検出
      OUT     Y332  ; RB IN562
8649  LD      L12  ; ﾚｰﾝ5下 M12選択中
      AND     L103  ; ﾚｰﾝ2下(M12)取出し
      ANI     L104  ; ﾚｰﾝ3上(M12)取出し
      LD      L13  ; ﾚｰﾝ5下 M10選択中
      AND     L109  ; ﾚｰﾝ5下(中間)取出し
      ANI     L106  ; ﾚｰﾝ4上(中間)取出し
      ORB
      OR      M16  ; 教示ﾓｰﾄﾞ
      AND     M860  ; ｽﾄｯｶｰ取出し開始条件
      AND     T176  ; ﾚｰﾝ2下段(M12)切出し部ﾜｰｸ検出
      OUT     Y333  ; RB IN563
8660  LD      L4  ; ﾚｰﾝ6上 M12選択中
      AND     L104  ; ﾚｰﾝ3上(M12)取出し
      ANI     L105  ; ﾚｰﾝ3下(M12)取出し
      LD      L5  ; ﾚｰﾝ6上 M10選択中
      AND     L110  ; ﾚｰﾝ6上(中間)取出し
      ANI     L111  ; ﾚｰﾝ6下(中間)取出し
      ORB
      OR      M16  ; 教示ﾓｰﾄﾞ
      AND     M860  ; ｽﾄｯｶｰ取出し開始条件
      AND     T178  ; ﾚｰﾝ3上段(M12)切出し部ﾜｰｸ検出
      OUT     Y334  ; RB IN564
8671  LD      L14  ; ﾚｰﾝ6下 M12選択中
      AND     L105  ; ﾚｰﾝ3下(M12)取出し
      ANI     L132  ; ﾚｰﾝ4上(中間)取出し
      LD      L15  ; ﾚｰﾝ6下 M10選択中
      AND     L111  ; ﾚｰﾝ6下(中間)取出し
      ANI     L108  ; ﾚｰﾝ5上(中間)取出し
      ORB
      OR      M16  ; 教示ﾓｰﾄﾞ
      AND     M860  ; ｽﾄｯｶｰ取出し開始条件
      AND     T180  ; ﾚｰﾝ3下段(M12)切出し部ﾜｰｸ検出
      OUT     Y335  ; RB IN565
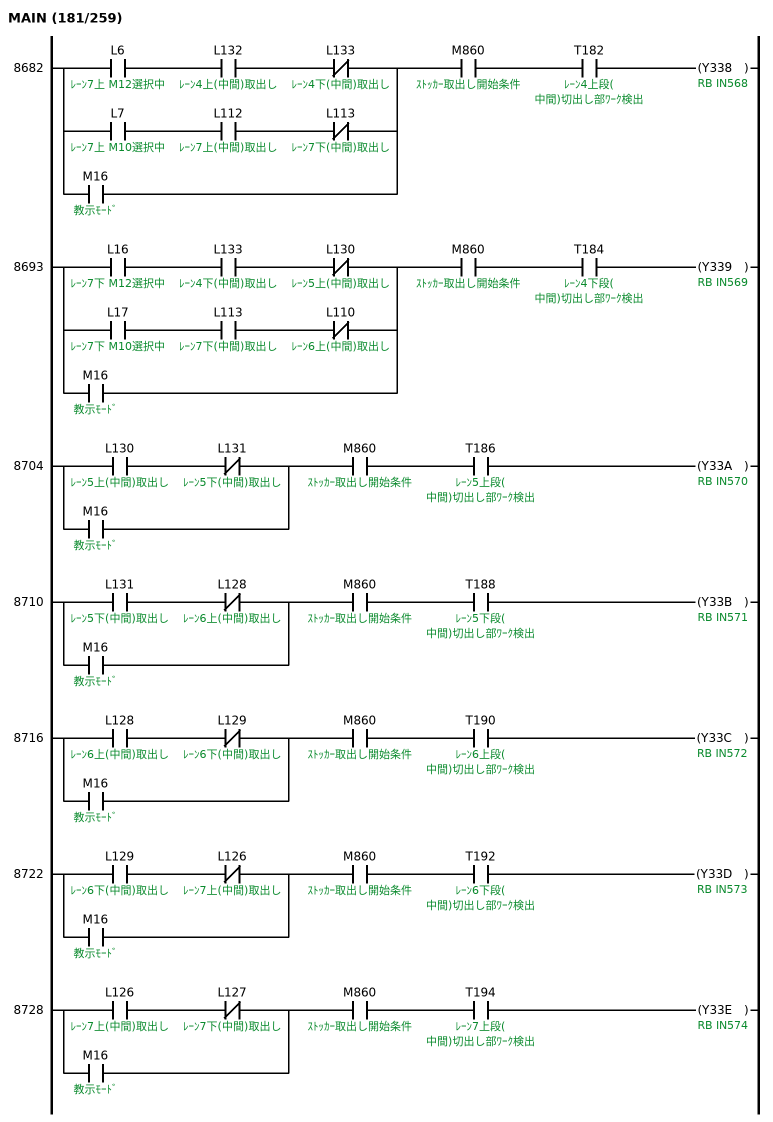
8682  LD      L6  ; ﾚｰﾝ7上 M12選択中
      AND     L132  ; ﾚｰﾝ4上(中間)取出し
      ANI     L133  ; ﾚｰﾝ4下(中間)取出し
      LD      L7  ; ﾚｰﾝ7上 M10選択中
      AND     L112  ; ﾚｰﾝ7上(中間)取出し
      ANI     L113  ; ﾚｰﾝ7下(中間)取出し
      ORB
      OR      M16  ; 教示ﾓｰﾄﾞ
      AND     M860  ; ｽﾄｯｶｰ取出し開始条件
      AND     T182  ; ﾚｰﾝ4上段(中間)切出し部ﾜｰｸ検出
      OUT     Y338  ; RB IN568
8693  LD      L16  ; ﾚｰﾝ7下 M12選択中
      AND     L133  ; ﾚｰﾝ4下(中間)取出し
      ANI     L130  ; ﾚｰﾝ5上(中間)取出し
      LD      L17  ; ﾚｰﾝ7下 M10選択中
      AND     L113  ; ﾚｰﾝ7下(中間)取出し
      ANI     L110  ; ﾚｰﾝ6上(中間)取出し
      ORB
      OR      M16  ; 教示ﾓｰﾄﾞ
      AND     M860  ; ｽﾄｯｶｰ取出し開始条件
      AND     T184  ; ﾚｰﾝ4下段(中間)切出し部ﾜｰｸ検出
      OUT     Y339  ; RB IN569
8704  LD      L130  ; ﾚｰﾝ5上(中間)取出し
      ANI     L131  ; ﾚｰﾝ5下(中間)取出し
      OR      M16  ; 教示ﾓｰﾄﾞ
      AND     M860  ; ｽﾄｯｶｰ取出し開始条件
      AND     T186  ; ﾚｰﾝ5上段(中間)切出し部ﾜｰｸ検出
      OUT     Y33A  ; RB IN570
8710  LD      L131  ; ﾚｰﾝ5下(中間)取出し
      ANI     L128  ; ﾚｰﾝ6上(中間)取出し
      OR      M16  ; 教示ﾓｰﾄﾞ
      AND     M860  ; ｽﾄｯｶｰ取出し開始条件
      AND     T188  ; ﾚｰﾝ5下段(中間)切出し部ﾜｰｸ検出
      OUT     Y33B  ; RB IN571
8716  LD      L128  ; ﾚｰﾝ6上(中間)取出し
      ANI     L129  ; ﾚｰﾝ6下(中間)取出し
      OR      M16  ; 教示ﾓｰﾄﾞ
      AND     M860  ; ｽﾄｯｶｰ取出し開始条件
      AND     T190  ; ﾚｰﾝ6上段(中間)切出し部ﾜｰｸ検出
      OUT     Y33C  ; RB IN572
8722  LD      L129  ; ﾚｰﾝ6下(中間)取出し
      ANI     L126  ; ﾚｰﾝ7上(中間)取出し
      OR      M16  ; 教示ﾓｰﾄﾞ
      AND     M860  ; ｽﾄｯｶｰ取出し開始条件
      AND     T192  ; ﾚｰﾝ6下段(中間)切出し部ﾜｰｸ検出
      OUT     Y33D  ; RB IN573
8728  LD      L126  ; ﾚｰﾝ7上(中間)取出し
      ANI     L127  ; ﾚｰﾝ7下(中間)取出し
      OR      M16  ; 教示ﾓｰﾄﾞ
      AND     M860  ; ｽﾄｯｶｰ取出し開始条件
      AND     T194  ; ﾚｰﾝ7上段(中間)切出し部ﾜｰｸ検出
      OUT     Y33E  ; RB IN574
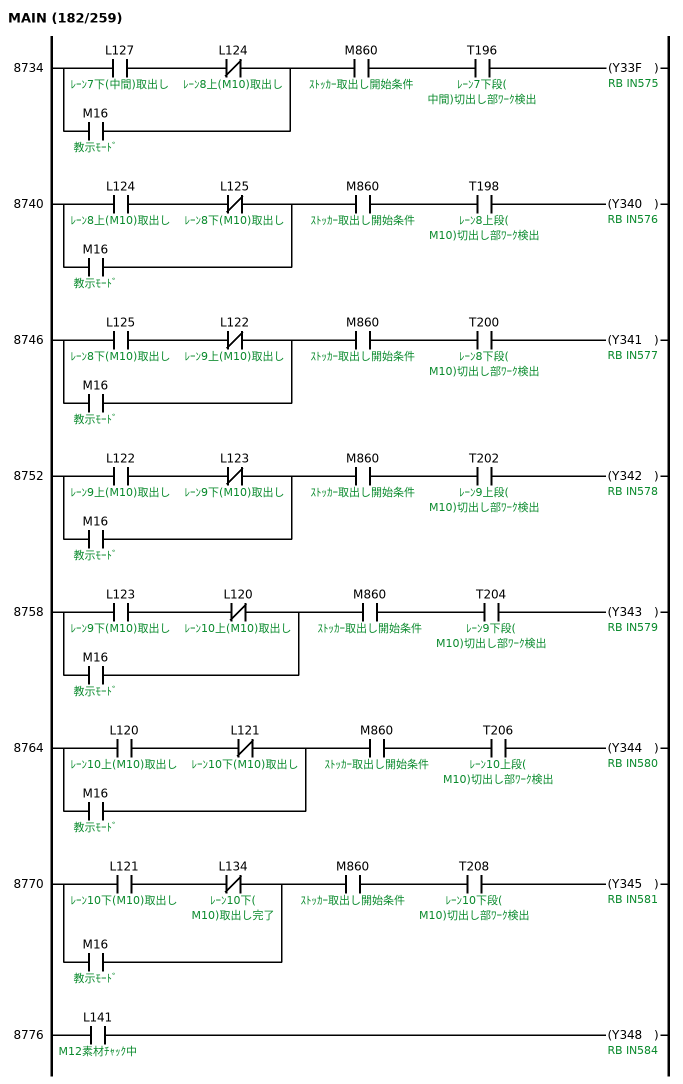
8734  LD      L127  ; ﾚｰﾝ7下(中間)取出し
      ANI     L124  ; ﾚｰﾝ8上(M10)取出し
      OR      M16  ; 教示ﾓｰﾄﾞ
      AND     M860  ; ｽﾄｯｶｰ取出し開始条件
      AND     T196  ; ﾚｰﾝ7下段(中間)切出し部ﾜｰｸ検出
      OUT     Y33F  ; RB IN575
8740  LD      L124  ; ﾚｰﾝ8上(M10)取出し
      ANI     L125  ; ﾚｰﾝ8下(M10)取出し
      OR      M16  ; 教示ﾓｰﾄﾞ
      AND     M860  ; ｽﾄｯｶｰ取出し開始条件
      AND     T198  ; ﾚｰﾝ8上段(M10)切出し部ﾜｰｸ検出
      OUT     Y340  ; RB IN576
8746  LD      L125  ; ﾚｰﾝ8下(M10)取出し
      ANI     L122  ; ﾚｰﾝ9上(M10)取出し
      OR      M16  ; 教示ﾓｰﾄﾞ
      AND     M860  ; ｽﾄｯｶｰ取出し開始条件
      AND     T200  ; ﾚｰﾝ8下段(M10)切出し部ﾜｰｸ検出
      OUT     Y341  ; RB IN577
8752  LD      L122  ; ﾚｰﾝ9上(M10)取出し
      ANI     L123  ; ﾚｰﾝ9下(M10)取出し
      OR      M16  ; 教示ﾓｰﾄﾞ
      AND     M860  ; ｽﾄｯｶｰ取出し開始条件
      AND     T202  ; ﾚｰﾝ9上段(M10)切出し部ﾜｰｸ検出
      OUT     Y342  ; RB IN578
8758  LD      L123  ; ﾚｰﾝ9下(M10)取出し
      ANI     L120  ; ﾚｰﾝ10上(M10)取出し
      OR      M16  ; 教示ﾓｰﾄﾞ
      AND     M860  ; ｽﾄｯｶｰ取出し開始条件
      AND     T204  ; ﾚｰﾝ9下段(M10)切出し部ﾜｰｸ検出
      OUT     Y343  ; RB IN579
8764  LD      L120  ; ﾚｰﾝ10上(M10)取出し
      ANI     L121  ; ﾚｰﾝ10下(M10)取出し
      OR      M16  ; 教示ﾓｰﾄﾞ
      AND     M860  ; ｽﾄｯｶｰ取出し開始条件
      AND     T206  ; ﾚｰﾝ10上段(M10)切出し部ﾜｰｸ検出
      OUT     Y344  ; RB IN580
8770  LD      L121  ; ﾚｰﾝ10下(M10)取出し
      ANI     L134  ; ﾚｰﾝ10下(M10)取出し完了
      OR      M16  ; 教示ﾓｰﾄﾞ
      AND     M860  ; ｽﾄｯｶｰ取出し開始条件
      AND     T208  ; ﾚｰﾝ10下段(M10)切出し部ﾜｰｸ検出
      OUT     Y345  ; RB IN581
8776  LD      L141  ; M12素材ﾁｬｯｸ中
      OUT     Y348  ; RB IN584
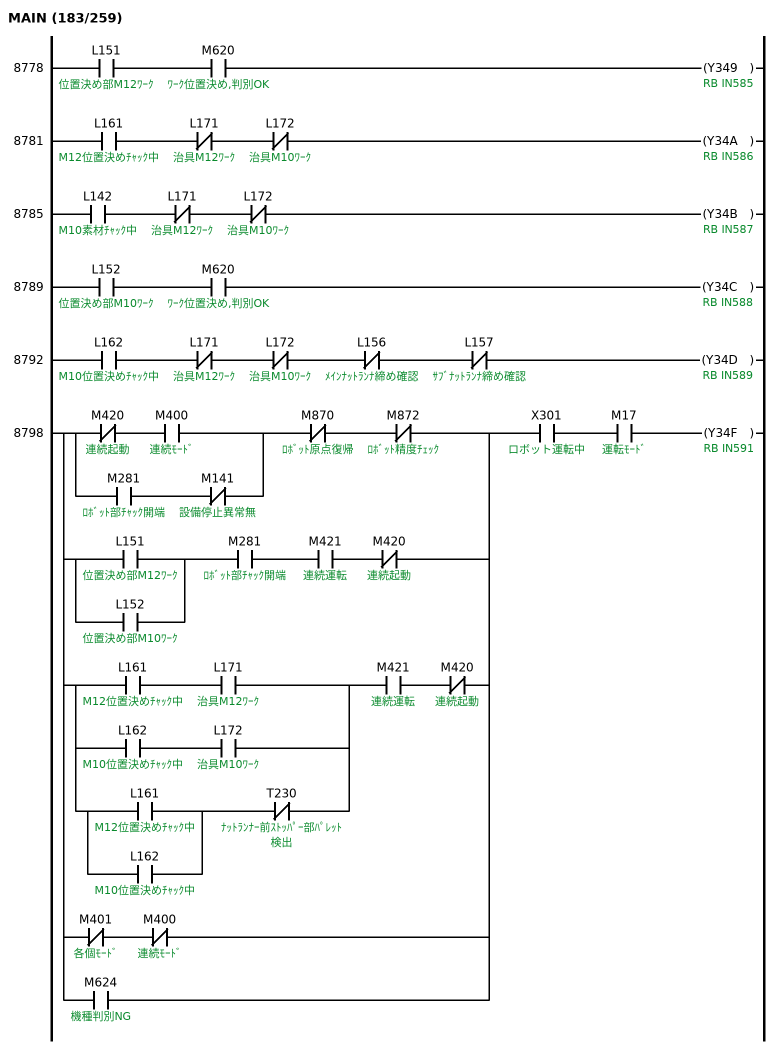
8778  LD      L151  ; 位置決め部M12ﾜｰｸ
      AND     M620  ; ﾜｰｸ位置決め,判別OK
      OUT     Y349  ; RB IN585
8781  LD      L161  ; M12位置決めﾁｬｯｸ中
      ANI     L171  ; 治具M12ﾜｰｸ
      ANI     L172  ; 治具M10ﾜｰｸ
      OUT     Y34A  ; RB IN586
8785  LD      L142  ; M10素材ﾁｬｯｸ中
      ANI     L171  ; 治具M12ﾜｰｸ
      ANI     L172  ; 治具M10ﾜｰｸ
      OUT     Y34B  ; RB IN587
8789  LD      L152  ; 位置決め部M10ﾜｰｸ
      AND     M620  ; ﾜｰｸ位置決め,判別OK
      OUT     Y34C  ; RB IN588
8792  LD      L162  ; M10位置決めﾁｬｯｸ中
      ANI     L171  ; 治具M12ﾜｰｸ
      ANI     L172  ; 治具M10ﾜｰｸ
      ANI     L156  ; ﾒｲﾝﾅｯﾄﾗﾝﾅ締め確認
      ANI     L157  ; ｻﾌﾞﾅｯﾄﾗﾝﾅ締め確認
      OUT     Y34D  ; RB IN589
8798  LDI     M420  ; 連続起動
      AND     M400  ; 連続ﾓｰﾄﾞ
      LD      M281  ; ﾛﾎﾞｯﾄ部ﾁｬｯｸ開端
      ANI     M141  ; 設備停止異常無
      ORB
      ANI     M870  ; ﾛﾎﾞｯﾄ原点復帰
      ANI     M872  ; ﾛﾎﾞｯﾄ精度ﾁｪｯｸ
      LD      L151  ; 位置決め部M12ﾜｰｸ
      OR      L152  ; 位置決め部M10ﾜｰｸ
      AND     M281  ; ﾛﾎﾞｯﾄ部ﾁｬｯｸ開端
      AND     M421  ; 連続運転
      ANI     M420  ; 連続起動
      ORB
      LD      L161  ; M12位置決めﾁｬｯｸ中
      AND     L171  ; 治具M12ﾜｰｸ
      LD      L162  ; M10位置決めﾁｬｯｸ中
      AND     L172  ; 治具M10ﾜｰｸ
      ORB
      LD      L161  ; M12位置決めﾁｬｯｸ中
      OR      L162  ; M10位置決めﾁｬｯｸ中
      ANI     T230  ; ﾅｯﾄﾗﾝﾅｰ前ｽﾄｯﾊﾟｰ部ﾊﾟﾚｯﾄ検出
      ORB
      AND     M421  ; 連続運転
      ANI     M420  ; 連続起動
      ORB
      LDI     M401  ; 各個ﾓｰﾄﾞ
      ANI     M400  ; 連続ﾓｰﾄﾞ
      ORB
      OR      M624  ; 機種判別NG
      AND     X301  ; ロボット運転中
      AND     M17  ; 運転ﾓｰﾄﾞ
      OUT     Y34F  ; RB IN591
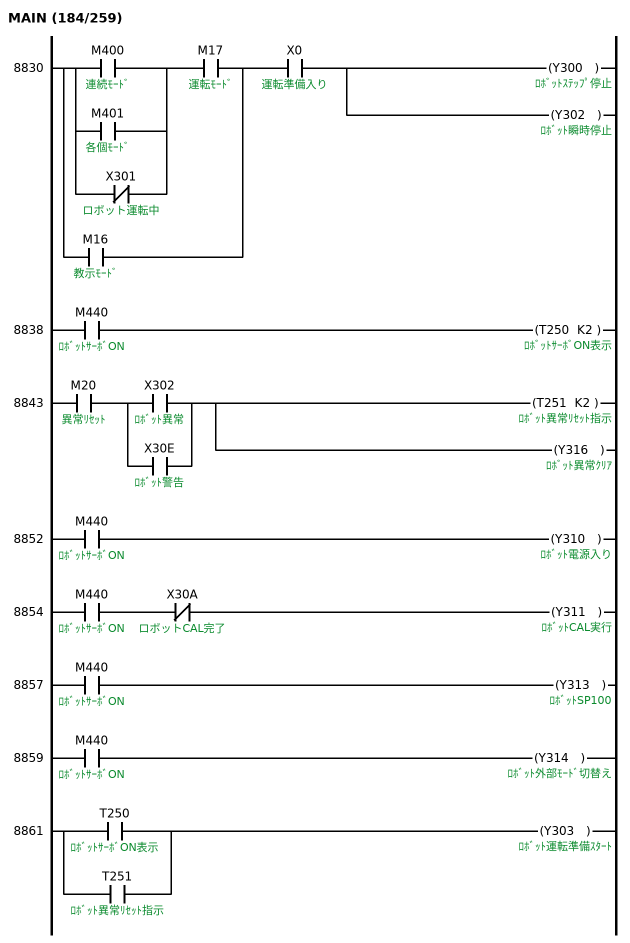
8830  LD      M400  ; 連続ﾓｰﾄﾞ
      OR      M401  ; 各個ﾓｰﾄﾞ
      ORI     X301  ; ロボット運転中
      AND     M17  ; 運転ﾓｰﾄﾞ
      OR      M16  ; 教示ﾓｰﾄﾞ
      AND     X0  ; 運転準備入り
      OUT     Y300  ; ﾛﾎﾞｯﾄｽﾃｯﾌﾟ停止
      OUT     Y302  ; ﾛﾎﾞｯﾄ瞬時停止
8838  LD      M440  ; ﾛﾎﾞｯﾄｻｰﾎﾞON
      OUT     T250 K2  ; ﾛﾎﾞｯﾄｻｰﾎﾞON表示
8843  LD      M20  ; 異常ﾘｾｯﾄ
      LD      X302  ; ﾛﾎﾞｯﾄ異常
      OR      X30E  ; ﾛﾎﾞｯﾄ警告
      ANB
      OUT     T251 K2  ; ﾛﾎﾞｯﾄ異常ﾘｾｯﾄ指示
      OUT     Y316  ; ﾛﾎﾞｯﾄ異常ｸﾘｱ
8852  LD      M440  ; ﾛﾎﾞｯﾄｻｰﾎﾞON
      OUT     Y310  ; ﾛﾎﾞｯﾄ電源入り
8854  LD      M440  ; ﾛﾎﾞｯﾄｻｰﾎﾞON
      ANI     X30A  ; ロボットCAL完了
      OUT     Y311  ; ﾛﾎﾞｯﾄCAL実行
8857  LD      M440  ; ﾛﾎﾞｯﾄｻｰﾎﾞON
      OUT     Y313  ; ﾛﾎﾞｯﾄSP100
8859  LD      M440  ; ﾛﾎﾞｯﾄｻｰﾎﾞON
      OUT     Y314  ; ﾛﾎﾞｯﾄ外部ﾓｰﾄﾞ切替え
8861  LD      T250  ; ﾛﾎﾞｯﾄｻｰﾎﾞON表示
      OR      T251  ; ﾛﾎﾞｯﾄ異常ﾘｾｯﾄ指示
      OUT     Y303  ; ﾛﾎﾞｯﾄ運転準備ｽﾀｰﾄ
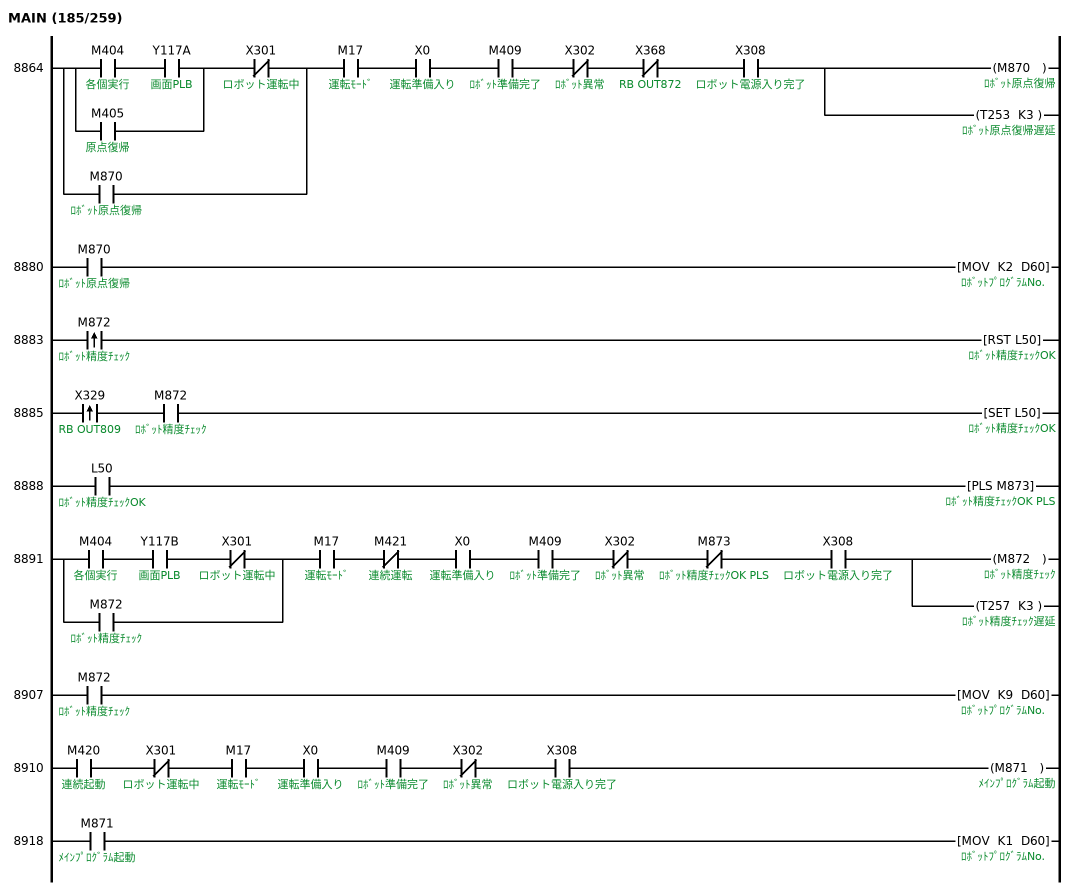
8864  LD      M404  ; 各個実行
      AND     Y117A  ; 画面PLB
      OR      M405  ; 原点復帰
      ANI     X301  ; ロボット運転中
      OR      M870  ; ﾛﾎﾞｯﾄ原点復帰
      AND     M17  ; 運転ﾓｰﾄﾞ
      AND     X0  ; 運転準備入り
      AND     M409  ; ﾛﾎﾞｯﾄ準備完了
      ANI     X302  ; ﾛﾎﾞｯﾄ異常
      ANI     X368  ; RB OUT872
      AND     X308  ; ロボット電源入り完了
      OUT     M870  ; ﾛﾎﾞｯﾄ原点復帰
      OUT     T253 K3  ; ﾛﾎﾞｯﾄ原点復帰遅延
8880  LD      M870  ; ﾛﾎﾞｯﾄ原点復帰
      MOV     K2 D60  ; ﾛﾎﾞｯﾄﾌﾟﾛｸﾞﾗﾑNo.
8883  LDP     M872  ; ﾛﾎﾞｯﾄ精度ﾁｪｯｸ
      RST     L50  ; ﾛﾎﾞｯﾄ精度ﾁｪｯｸOK
8885  LDP     X329  ; RB OUT809
      AND     M872  ; ﾛﾎﾞｯﾄ精度ﾁｪｯｸ
      SET     L50  ; ﾛﾎﾞｯﾄ精度ﾁｪｯｸOK
8888  LD      L50  ; ﾛﾎﾞｯﾄ精度ﾁｪｯｸOK
      PLS     M873  ; ﾛﾎﾞｯﾄ精度ﾁｪｯｸOK PLS
8891  LD      M404  ; 各個実行
      AND     Y117B  ; 画面PLB
      ANI     X301  ; ロボット運転中
      OR      M872  ; ﾛﾎﾞｯﾄ精度ﾁｪｯｸ
      AND     M17  ; 運転ﾓｰﾄﾞ
      ANI     M421  ; 連続運転
      AND     X0  ; 運転準備入り
      AND     M409  ; ﾛﾎﾞｯﾄ準備完了
      ANI     X302  ; ﾛﾎﾞｯﾄ異常
      ANI     M873  ; ﾛﾎﾞｯﾄ精度ﾁｪｯｸOK PLS
      AND     X308  ; ロボット電源入り完了
      OUT     M872  ; ﾛﾎﾞｯﾄ精度ﾁｪｯｸ
      OUT     T257 K3  ; ﾛﾎﾞｯﾄ精度ﾁｪｯｸ遅延
8907  LD      M872  ; ﾛﾎﾞｯﾄ精度ﾁｪｯｸ
      MOV     K9 D60
8910  LD      M420  ; 連続起動
      ANI     X301  ; ロボット運転中
      AND     M17  ; 運転ﾓｰﾄﾞ
      AND     X0  ; 運転準備入り
      AND     M409  ; ﾛﾎﾞｯﾄ準備完了
      ANI     X302  ; ﾛﾎﾞｯﾄ異常
      AND     X308  ; ロボット電源入り完了
      OUT     M871  ; ﾒｲﾝﾌﾟﾛｸﾞﾗﾑ起動
8918  LD      M871  ; ﾒｲﾝﾌﾟﾛｸﾞﾗﾑ起動
      MOV     K1 D60
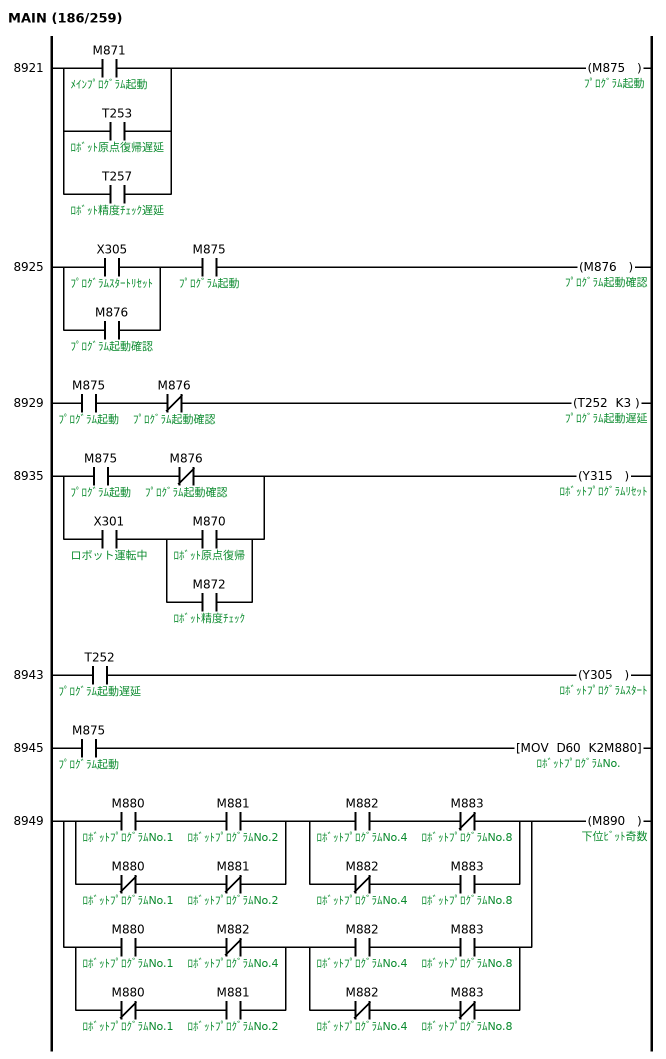
8921  LD      M871  ; ﾒｲﾝﾌﾟﾛｸﾞﾗﾑ起動
      OR      T253  ; ﾛﾎﾞｯﾄ原点復帰遅延
      OR      T257  ; ﾛﾎﾞｯﾄ精度ﾁｪｯｸ遅延
      OUT     M875  ; ﾌﾟﾛｸﾞﾗﾑ起動
8925  LD      X305  ; ﾌﾟﾛｸﾞﾗﾑｽﾀｰﾄﾘｾｯﾄ
      OR      M876  ; ﾌﾟﾛｸﾞﾗﾑ起動確認
      AND     M875  ; ﾌﾟﾛｸﾞﾗﾑ起動
      OUT     M876  ; ﾌﾟﾛｸﾞﾗﾑ起動確認
8929  LD      M875  ; ﾌﾟﾛｸﾞﾗﾑ起動
      ANI     M876  ; ﾌﾟﾛｸﾞﾗﾑ起動確認
      OUT     T252 K3  ; ﾌﾟﾛｸﾞﾗﾑ起動遅延
8935  LD      M875  ; ﾌﾟﾛｸﾞﾗﾑ起動
      ANI     M876  ; ﾌﾟﾛｸﾞﾗﾑ起動確認
      LD      X301  ; ロボット運転中
      LD      M870  ; ﾛﾎﾞｯﾄ原点復帰
      OR      M872  ; ﾛﾎﾞｯﾄ精度ﾁｪｯｸ
      ANB
      ORB
      OUT     Y315  ; ﾛﾎﾞｯﾄﾌﾟﾛｸﾞﾗﾑﾘｾｯﾄ
8943  LD      T252  ; ﾌﾟﾛｸﾞﾗﾑ起動遅延
      OUT     Y305  ; ﾛﾎﾞｯﾄﾌﾟﾛｸﾞﾗﾑｽﾀｰﾄ
8945  LD      M875  ; ﾌﾟﾛｸﾞﾗﾑ起動
      MOV     D60 K2M880  ; ﾛﾎﾞｯﾄﾌﾟﾛｸﾞﾗﾑNo.1
8949  LD      M880  ; ﾛﾎﾞｯﾄﾌﾟﾛｸﾞﾗﾑNo.1
      AND     M881  ; ﾛﾎﾞｯﾄﾌﾟﾛｸﾞﾗﾑNo.2
      LDI     M880  ; ﾛﾎﾞｯﾄﾌﾟﾛｸﾞﾗﾑNo.1
      ANI     M881  ; ﾛﾎﾞｯﾄﾌﾟﾛｸﾞﾗﾑNo.2
      ORB
      LD      M882  ; ﾛﾎﾞｯﾄﾌﾟﾛｸﾞﾗﾑNo.4
      ANI     M883  ; ﾛﾎﾞｯﾄﾌﾟﾛｸﾞﾗﾑNo.8
      LDI     M882  ; ﾛﾎﾞｯﾄﾌﾟﾛｸﾞﾗﾑNo.4
      AND     M883  ; ﾛﾎﾞｯﾄﾌﾟﾛｸﾞﾗﾑNo.8
      ORB
      ANB
      LD      M880  ; ﾛﾎﾞｯﾄﾌﾟﾛｸﾞﾗﾑNo.1
      ANI     M882  ; ﾛﾎﾞｯﾄﾌﾟﾛｸﾞﾗﾑNo.4
      LDI     M880  ; ﾛﾎﾞｯﾄﾌﾟﾛｸﾞﾗﾑNo.1
      AND     M881  ; ﾛﾎﾞｯﾄﾌﾟﾛｸﾞﾗﾑNo.2
      ORB
      LD      M882  ; ﾛﾎﾞｯﾄﾌﾟﾛｸﾞﾗﾑNo.4
      AND     M883  ; ﾛﾎﾞｯﾄﾌﾟﾛｸﾞﾗﾑNo.8
      LDI     M882  ; ﾛﾎﾞｯﾄﾌﾟﾛｸﾞﾗﾑNo.4
      ANI     M883  ; ﾛﾎﾞｯﾄﾌﾟﾛｸﾞﾗﾑNo.8
      ORB
      ANB
      ORB
      OUT     M890  ; 下位ﾋﾞｯﾄ奇数
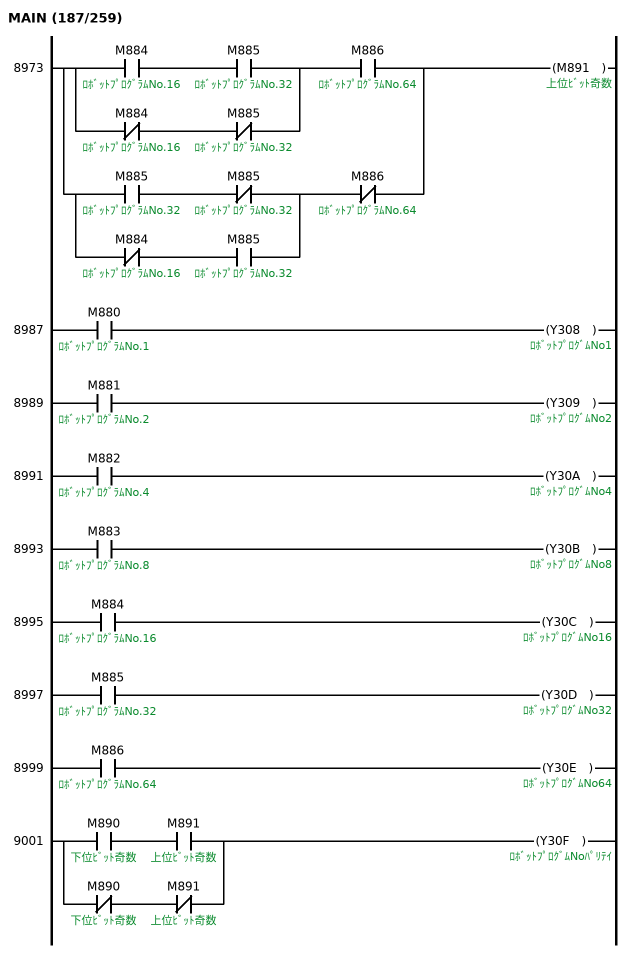
8973  LD      M884  ; ﾛﾎﾞｯﾄﾌﾟﾛｸﾞﾗﾑNo.16
      AND     M885  ; ﾛﾎﾞｯﾄﾌﾟﾛｸﾞﾗﾑNo.32
      LDI     M884  ; ﾛﾎﾞｯﾄﾌﾟﾛｸﾞﾗﾑNo.16
      ANI     M885  ; ﾛﾎﾞｯﾄﾌﾟﾛｸﾞﾗﾑNo.32
      ORB
      AND     M886  ; ﾛﾎﾞｯﾄﾌﾟﾛｸﾞﾗﾑNo.64
      LD      M885  ; ﾛﾎﾞｯﾄﾌﾟﾛｸﾞﾗﾑNo.32
      ANI     M885  ; ﾛﾎﾞｯﾄﾌﾟﾛｸﾞﾗﾑNo.32
      LDI     M884  ; ﾛﾎﾞｯﾄﾌﾟﾛｸﾞﾗﾑNo.16
      AND     M885  ; ﾛﾎﾞｯﾄﾌﾟﾛｸﾞﾗﾑNo.32
      ORB
      ANI     M886  ; ﾛﾎﾞｯﾄﾌﾟﾛｸﾞﾗﾑNo.64
      ORB
      OUT     M891  ; 上位ﾋﾞｯﾄ奇数
8987  LD      M880  ; ﾛﾎﾞｯﾄﾌﾟﾛｸﾞﾗﾑNo.1
      OUT     Y308  ; ﾛﾎﾞｯﾄﾌﾟﾛｸﾞﾑNo1
8989  LD      M881  ; ﾛﾎﾞｯﾄﾌﾟﾛｸﾞﾗﾑNo.2
      OUT     Y309  ; ﾛﾎﾞｯﾄﾌﾟﾛｸﾞﾑNo2
8991  LD      M882  ; ﾛﾎﾞｯﾄﾌﾟﾛｸﾞﾗﾑNo.4
      OUT     Y30A  ; ﾛﾎﾞｯﾄﾌﾟﾛｸﾞﾑNo4
8993  LD      M883  ; ﾛﾎﾞｯﾄﾌﾟﾛｸﾞﾗﾑNo.8
      OUT     Y30B  ; ﾛﾎﾞｯﾄﾌﾟﾛｸﾞﾑNo8
8995  LD      M884  ; ﾛﾎﾞｯﾄﾌﾟﾛｸﾞﾗﾑNo.16
      OUT     Y30C  ; ﾛﾎﾞｯﾄﾌﾟﾛｸﾞﾑNo16
8997  LD      M885  ; ﾛﾎﾞｯﾄﾌﾟﾛｸﾞﾗﾑNo.32
      OUT     Y30D  ; ﾛﾎﾞｯﾄﾌﾟﾛｸﾞﾑNo32
8999  LD      M886  ; ﾛﾎﾞｯﾄﾌﾟﾛｸﾞﾗﾑNo.64
      OUT     Y30E  ; ﾛﾎﾞｯﾄﾌﾟﾛｸﾞﾑNo64
9001  LD      M890  ; 下位ﾋﾞｯﾄ奇数
      AND     M891  ; 上位ﾋﾞｯﾄ奇数
      LDI     M890  ; 下位ﾋﾞｯﾄ奇数
      ANI     M891  ; 上位ﾋﾞｯﾄ奇数
      ORB
      OUT     Y30F  ; ﾛﾎﾞｯﾄﾌﾟﾛｸﾞﾑNoﾊﾟﾘﾃｲ
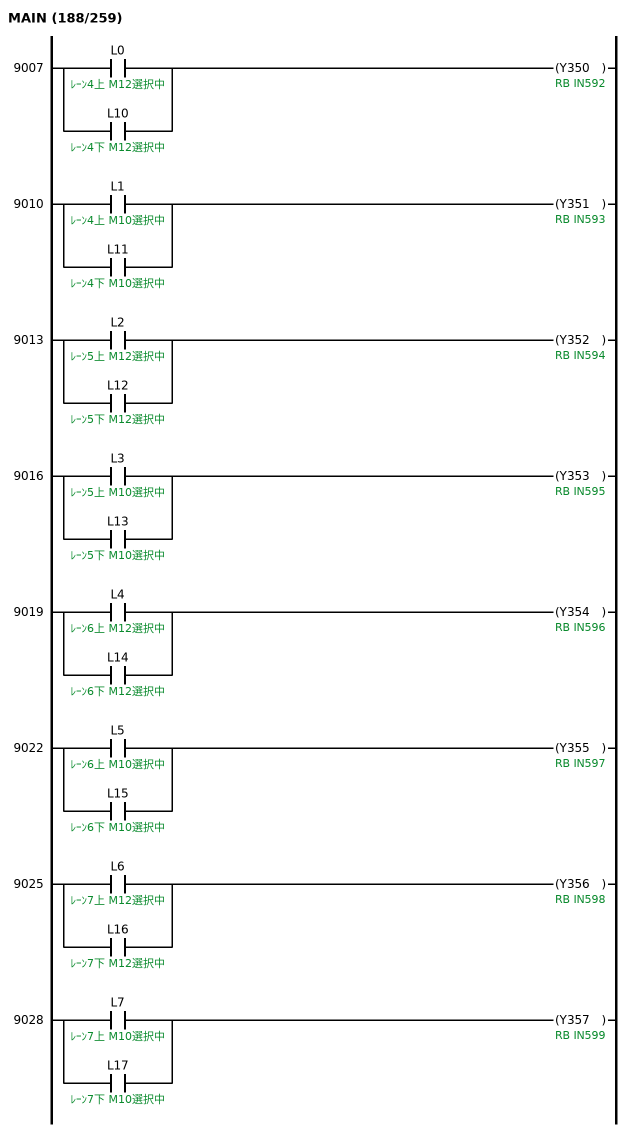
9007  LD      L0  ; ﾚｰﾝ4上 M12選択中
      OR      L10  ; ﾚｰﾝ4下 M12選択中
      OUT     Y350  ; RB IN592
9010  LD      L1  ; ﾚｰﾝ4上 M10選択中
      OR      L11  ; ﾚｰﾝ4下 M10選択中
      OUT     Y351  ; RB IN593
9013  LD      L2  ; ﾚｰﾝ5上 M12選択中
      OR      L12  ; ﾚｰﾝ5下 M12選択中
      OUT     Y352  ; RB IN594
9016  LD      L3  ; ﾚｰﾝ5上 M10選択中
      OR      L13  ; ﾚｰﾝ5下 M10選択中
      OUT     Y353  ; RB IN595
9019  LD      L4  ; ﾚｰﾝ6上 M12選択中
      OR      L14  ; ﾚｰﾝ6下 M12選択中
      OUT     Y354  ; RB IN596
9022  LD      L5  ; ﾚｰﾝ6上 M10選択中
      OR      L15  ; ﾚｰﾝ6下 M10選択中
      OUT     Y355  ; RB IN597
9025  LD      L6  ; ﾚｰﾝ7上 M12選択中
      OR      L16  ; ﾚｰﾝ7下 M12選択中
      OUT     Y356  ; RB IN598
9028  LD      L7  ; ﾚｰﾝ7上 M10選択中
      OR      L17  ; ﾚｰﾝ7下 M10選択中
      OUT     Y357  ; RB IN599
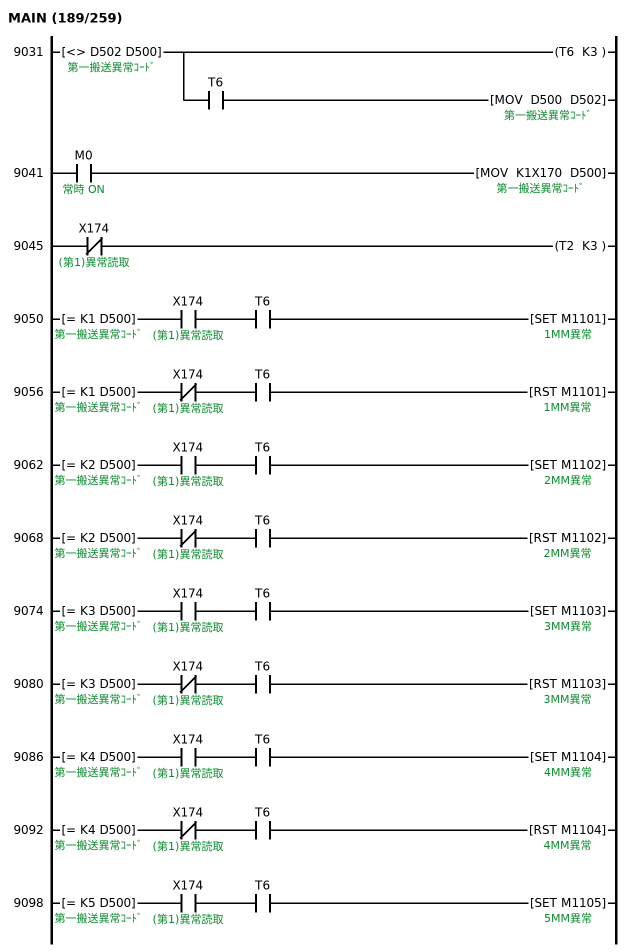
9031  LD<>    D502 D500  ; 第一搬送異常ｺｰﾄﾞ
      OUT     T6 K3
      AND     T6
      MOV     D500 D502
9041  LD      M0  ; 常時 ON
      MOV     K1X170 D500  ; (第1)異常ｺｰﾄﾞ1
9045  LDI     X174  ; (第1)異常読取
      OUT     T2 K3
9050  LD=     K1 D500  ; 第一搬送異常ｺｰﾄﾞ
      AND     X174  ; (第1)異常読取
      AND     T6
      SET     M1101  ; 1MM異常
9056  LD=     K1 D500  ; 第一搬送異常ｺｰﾄﾞ
      ANI     X174  ; (第1)異常読取
      AND     T6
      RST     M1101  ; 1MM異常
9062  LD=     K2 D500  ; 第一搬送異常ｺｰﾄﾞ
      AND     X174  ; (第1)異常読取
      AND     T6
      SET     M1102  ; 2MM異常
9068  LD=     K2 D500  ; 第一搬送異常ｺｰﾄﾞ
      ANI     X174  ; (第1)異常読取
      AND     T6
      RST     M1102  ; 2MM異常
9074  LD=     K3 D500  ; 第一搬送異常ｺｰﾄﾞ
      AND     X174  ; (第1)異常読取
      AND     T6
      SET     M1103  ; 3MM異常
9080  LD=     K3 D500  ; 第一搬送異常ｺｰﾄﾞ
      ANI     X174  ; (第1)異常読取
      AND     T6
      RST     M1103  ; 3MM異常
9086  LD=     K4 D500  ; 第一搬送異常ｺｰﾄﾞ
      AND     X174  ; (第1)異常読取
      AND     T6
      SET     M1104  ; 4MM異常
9092  LD=     K4 D500  ; 第一搬送異常ｺｰﾄﾞ
      ANI     X174  ; (第1)異常読取
      AND     T6
      RST     M1104  ; 4MM異常
9098  LD=     K5 D500  ; 第一搬送異常ｺｰﾄﾞ
      AND     X174  ; (第1)異常読取
      AND     T6
      SET     M1105  ; 5MM異常
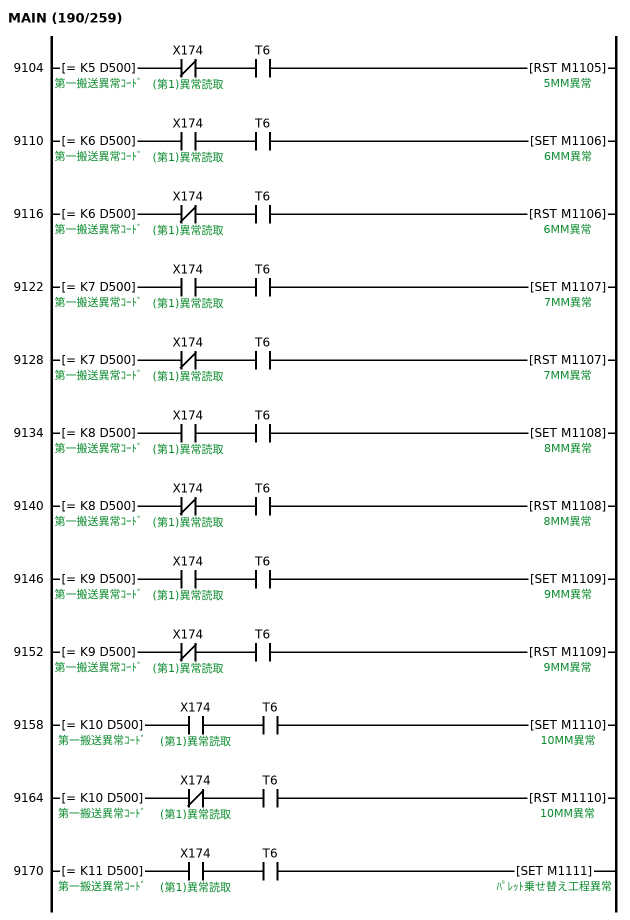
9104  LD=     K5 D500  ; 第一搬送異常ｺｰﾄﾞ
      ANI     X174  ; (第1)異常読取
      AND     T6
      RST     M1105  ; 5MM異常
9110  LD=     K6 D500  ; 第一搬送異常ｺｰﾄﾞ
      AND     X174  ; (第1)異常読取
      AND     T6
      SET     M1106  ; 6MM異常
9116  LD=     K6 D500  ; 第一搬送異常ｺｰﾄﾞ
      ANI     X174  ; (第1)異常読取
      AND     T6
      RST     M1106  ; 6MM異常
9122  LD=     K7 D500  ; 第一搬送異常ｺｰﾄﾞ
      AND     X174  ; (第1)異常読取
      AND     T6
      SET     M1107  ; 7MM異常
9128  LD=     K7 D500  ; 第一搬送異常ｺｰﾄﾞ
      ANI     X174  ; (第1)異常読取
      AND     T6
      RST     M1107  ; 7MM異常
9134  LD=     K8 D500  ; 第一搬送異常ｺｰﾄﾞ
      AND     X174  ; (第1)異常読取
      AND     T6
      SET     M1108  ; 8MM異常
9140  LD=     K8 D500  ; 第一搬送異常ｺｰﾄﾞ
      ANI     X174  ; (第1)異常読取
      AND     T6
      RST     M1108  ; 8MM異常
9146  LD=     K9 D500  ; 第一搬送異常ｺｰﾄﾞ
      AND     X174  ; (第1)異常読取
      AND     T6
      SET     M1109  ; 9MM異常
9152  LD=     K9 D500  ; 第一搬送異常ｺｰﾄﾞ
      ANI     X174  ; (第1)異常読取
      AND     T6
      RST     M1109  ; 9MM異常
9158  LD=     K10 D500  ; 第一搬送異常ｺｰﾄﾞ
      AND     X174  ; (第1)異常読取
      AND     T6
      SET     M1110  ; 10MM異常
9164  LD=     K10 D500  ; 第一搬送異常ｺｰﾄﾞ
      ANI     X174  ; (第1)異常読取
      AND     T6
      RST     M1110  ; 10MM異常
9170  LD=     K11 D500  ; 第一搬送異常ｺｰﾄﾞ
      AND     X174  ; (第1)異常読取
      AND     T6
      SET     M1111  ; ﾊﾟﾚｯﾄ乗せ替え工程異常
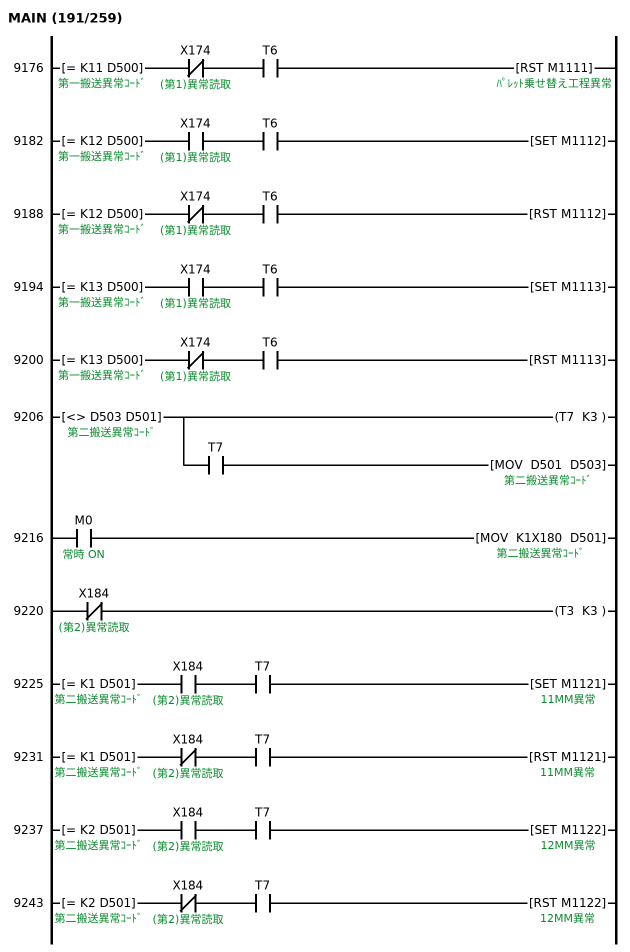
9176  LD=     K11 D500  ; 第一搬送異常ｺｰﾄﾞ
      ANI     X174  ; (第1)異常読取
      AND     T6
      RST     M1111  ; ﾊﾟﾚｯﾄ乗せ替え工程異常
9182  LD=     K12 D500  ; 第一搬送異常ｺｰﾄﾞ
      AND     X174  ; (第1)異常読取
      AND     T6
      SET     M1112
9188  LD=     K12 D500  ; 第一搬送異常ｺｰﾄﾞ
      ANI     X174  ; (第1)異常読取
      AND     T6
      RST     M1112
9194  LD=     K13 D500  ; 第一搬送異常ｺｰﾄﾞ
      AND     X174  ; (第1)異常読取
      AND     T6
      SET     M1113
9200  LD=     K13 D500  ; 第一搬送異常ｺｰﾄﾞ
      ANI     X174  ; (第1)異常読取
      AND     T6
      RST     M1113
9206  LD<>    D503 D501  ; 第二搬送異常ｺｰﾄﾞ
      OUT     T7 K3
      AND     T7
      MOV     D501 D503
9216  LD      M0  ; 常時 ON
      MOV     K1X180 D501  ; (第2)異常ｺｰﾄﾞ1
9220  LDI     X184  ; (第2)異常読取
      OUT     T3 K3
9225  LD=     K1 D501  ; 第二搬送異常ｺｰﾄﾞ
      AND     X184  ; (第2)異常読取
      AND     T7
      SET     M1121  ; 11MM異常
9231  LD=     K1 D501  ; 第二搬送異常ｺｰﾄﾞ
      ANI     X184  ; (第2)異常読取
      AND     T7
      RST     M1121  ; 11MM異常
9237  LD=     K2 D501  ; 第二搬送異常ｺｰﾄﾞ
      AND     X184  ; (第2)異常読取
      AND     T7
      SET     M1122  ; 12MM異常
9243  LD=     K2 D501  ; 第二搬送異常ｺｰﾄﾞ
      ANI     X184  ; (第2)異常読取
      AND     T7
      RST     M1122  ; 12MM異常
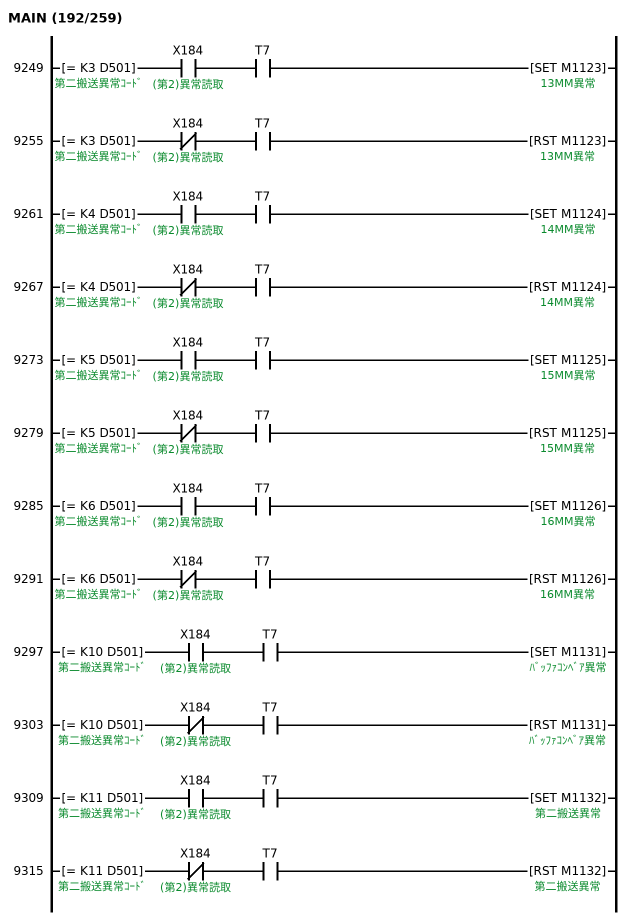
9249  LD=     K3 D501  ; 第二搬送異常ｺｰﾄﾞ
      AND     X184  ; (第2)異常読取
      AND     T7
      SET     M1123  ; 13MM異常
9255  LD=     K3 D501  ; 第二搬送異常ｺｰﾄﾞ
      ANI     X184  ; (第2)異常読取
      AND     T7
      RST     M1123  ; 13MM異常
9261  LD=     K4 D501  ; 第二搬送異常ｺｰﾄﾞ
      AND     X184  ; (第2)異常読取
      AND     T7
      SET     M1124  ; 14MM異常
9267  LD=     K4 D501  ; 第二搬送異常ｺｰﾄﾞ
      ANI     X184  ; (第2)異常読取
      AND     T7
      RST     M1124  ; 14MM異常
9273  LD=     K5 D501  ; 第二搬送異常ｺｰﾄﾞ
      AND     X184  ; (第2)異常読取
      AND     T7
      SET     M1125  ; 15MM異常
9279  LD=     K5 D501  ; 第二搬送異常ｺｰﾄﾞ
      ANI     X184  ; (第2)異常読取
      AND     T7
      RST     M1125  ; 15MM異常
9285  LD=     K6 D501  ; 第二搬送異常ｺｰﾄﾞ
      AND     X184  ; (第2)異常読取
      AND     T7
      SET     M1126  ; 16MM異常
9291  LD=     K6 D501  ; 第二搬送異常ｺｰﾄﾞ
      ANI     X184  ; (第2)異常読取
      AND     T7
      RST     M1126  ; 16MM異常
9297  LD=     K10 D501  ; 第二搬送異常ｺｰﾄﾞ
      AND     X184  ; (第2)異常読取
      AND     T7
      SET     M1131  ; ﾊﾞｯﾌｧｺﾝﾍﾞｱ異常
9303  LD=     K10 D501  ; 第二搬送異常ｺｰﾄﾞ
      ANI     X184  ; (第2)異常読取
      AND     T7
      RST     M1131  ; ﾊﾞｯﾌｧｺﾝﾍﾞｱ異常
9309  LD=     K11 D501  ; 第二搬送異常ｺｰﾄﾞ
      AND     X184  ; (第2)異常読取
      AND     T7
      SET     M1132  ; 第二搬送異常
9315  LD=     K11 D501  ; 第二搬送異常ｺｰﾄﾞ
      ANI     X184  ; (第2)異常読取
      AND     T7
      RST     M1132  ; 第二搬送異常
